LIN {X 0,Y 488.808,Z 370.599,A -85,B 0,C 180,E1 -6488.267,E2 -6488.267} C_VEL
LIN {X 0,Y 488.82,Z 370.594,A -85,B 0,C 180,E1 -6491.612,E2 -6491.612} C_VEL
LIN {X 0,Y 488.751,Z 370.602,A -85,B 0,C 180,E1 -6495.001,E2 -6495.001} C_VEL
LIN {X 0,Y 488.744,Z 370.605,A -85,B 0,C 180,E1 -6498.443,E2 -6498.443} C_VEL
LIN {X 0,Y 488.732,Z 370.603,A -85,B 0,C 180,E1 -6501.07,E2 -6501.07} C_VEL
LIN {X 0,Y 488.706,Z 370.612,A -85,B 0,C 180,E1 -6503.745,E2 -6503.745} C_VEL
LIN {X 0,Y 488.789,Z 370.596,A -85,B 0,C 180,E1 -6506.946,E2 -6506.946} C_VEL
LIN {X 0,Y 488.71,Z 370.607,A -85,B 0,C 180,E1 -6510.366,E2 -6510.366} C_VEL
LIN {X 0,Y 488.727,Z 370.609,A -85,B 0,C 180,E1 -6513.485,E2 -6513.485} C_VEL
LIN {X 0,Y 488.681,Z 370.609,A -85,B 0,C 180,E1 -6516.357,E2 -6516.357} C_VEL
LIN {X 0,Y 488.694,Z 370.613,A -85,B 0,C 180,E1 -6519.255,E2 -6519.255} C_VEL
LIN {X 0,Y 488.716,Z 370.609,A -85,B 0,C 180,E1 -6521.603,E2 -6521.603} C_VEL
LIN {X 0,Y 488.705,Z 370.608,A -85,B 0,C 180,E1 -6524.802,E2 -6524.802} C_VEL
LIN {X 0,Y 488.689,Z 370.612,A -85,B 0,C 180,E1 -6527.476,E2 -6527.476} C_VEL
LIN {X 0,Y 488.727,Z 370.605,A -85,B 0,C 180,E1 -6529.678,E2 -6529.678} C_VEL
LIN {X 0,Y 488.678,Z 370.615,A -85,B 0,C 180,E1 -6532.843,E2 -6532.843} C_VEL
LIN {X 0,Y 488.731,Z 370.604,A -85,B 0,C 180,E1 -6535.889,E2 -6535.889} C_VEL
LIN {X 0,Y 488.715,Z 370.612,A -85,B 0,C 180,E1 -6538.823,E2 -6538.823} C_VEL
LIN {X 0,Y 488.745,Z 370.603,A -85,B 0,C 180,E1 -6541.673,E2 -6541.673} C_VEL
LIN {X 0,Y 488.752,Z 370.607,A -85,B 0,C 180,E1 -6544.446,E2 -6544.446} C_VEL
LIN {X 0,Y 488.799,Z 370.776,A -85,B 0,C 180,E1 -6544.889,E2 -6544.889} C_VEL
LIN {X 0,Y 490.72,Z 381.32,A -85,B 0,C 180,E1 -6546.858,E2 -6546.858} C_VEL
LIN {X 0,Y 490.125,Z 397.445,A -85,B 0,C 180,E1 -6549.653,E2 -6549.653} C_VEL
LIN {X 0,Y 489.515,Z 415.125,A -85,B 0,C 180,E1 -6552.669,E2 -6552.669} C_VEL
LIN {X 0,Y 489.298,Z 421.438,A -85,B 0,C 180,E1 -6553.737,E2 -6553.737} C_VEL
LIN {X 0,Y 491.719,Z 437.9,A -85,B 0,C 180,E1 -6554.068,E2 -6554.068} C_VEL
LIN {X 0,Y 491.078,Z 529.428,A -85,B 0,C 180,E1 -6555.444,E2 -6555.444} C_VEL
LIN {X 0,Y 490.774,Z 542.701,A -85,B 0,C 180,E1 -6555.806,E2 -6555.806} C_VEL
LIN {X 0,Y 490.402,Z 555.445,A -85,B 0,C 180,E1 -6556.323,E2 -6556.323} C_VEL
LIN {X 0,Y 490.037,Z 567.098,A -85,B 0,C 180,E1 -6556.967,E2 -6556.967} C_VEL
LIN {X 0,Y 489.578,Z 578.466,A -85,B 0,C 180,E1 -6557.777,E2 -6557.777} C_VEL
LIN {X 0,Y 489.234,Z 588.982,A -85,B 0,C 180,E1 -6558.714,E2 -6558.714} C_VEL
LIN {X 0,Y 488.855,Z 597.575,A -85,B 0,C 180,E1 -6559.649,E2 -6559.649} C_VEL
LIN {X 0,Y 488.555,Z 605.502,A -85,B 0,C 180,E1 -6560.688,E2 -6560.688} C_VEL
LIN {X 0,Y 488.289,Z 613.245,A -85,B 0,C 180,E1 -6561.934,E2 -6561.934} C_VEL
LIN {X 0,Y 488.068,Z 620.369,A -85,B 0,C 180,E1 -6563.386,E2 -6563.386} C_VEL
LIN {X 0,Y 488.022,Z 625.112,A -85,B 0,C 180,E1 -6564.63,E2 -6564.63} C_VEL
LIN {X 0,Y 487.927,Z 628.733,A -85,B 0,C 180,E1 -6565.871,E2 -6565.871} C_VEL
LIN {X 0,Y 487.964,Z 630.602,A -85,B 0,C 180,E1 -6566.698,E2 -6566.698} C_VEL
LIN {X 0,Y 487.908,Z 632.001,A -85,B 0,C 180,E1 -6567.524,E2 -6567.524} C_VEL
LIN {X 0,Y 487.89,Z 632.998,A -85,B 0,C 180,E1 -6568.35,E2 -6568.35} C_VEL
LIN {X 0,Y 487.819,Z 633.817,A -85,B 0,C 180,E1 -6570.001,E2 -6570.001} C_VEL
LIN {X 0,Y 487.891,Z 632.984,A -85,B 0,C 180,E1 -6571.652,E2 -6571.652} C_VEL
LIN {X 0,Y 487.909,Z 631.98,A -85,B 0,C 180,E1 -6572.478,E2 -6572.478} C_VEL
LIN {X 0,Y 487.965,Z 630.574,A -85,B 0,C 180,E1 -6573.304,E2 -6573.304} C_VEL
LIN {X 0,Y 487.921,Z 627.615,A -85,B 0,C 180,E1 -6574.545,E2 -6574.545} C_VEL
LIN {X 0,Y 488.033,Z 623.616,A -85,B 0,C 180,E1 -6575.787,E2 -6575.787} C_VEL
LIN {X 0,Y 488.184,Z 617.461,A -85,B 0,C 180,E1 -6577.238,E2 -6577.238} C_VEL
LIN {X 0,Y 488.365,Z 610.737,A -85,B 0,C 180,E1 -6578.483,E2 -6578.483} C_VEL
LIN {X 0,Y 488.663,Z 602.397,A -85,B 0,C 180,E1 -6579.73,E2 -6579.73} C_VEL
LIN {X 0,Y 489.003,Z 593.832,A -85,B 0,C 180,E1 -6580.769,E2 -6580.769} C_VEL
LIN {X 0,Y 489.456,Z 583.255,A -85,B 0,C 180,E1 -6581.808,E2 -6581.808} C_VEL
LIN {X 0,Y 489.761,Z 572.902,A -85,B 0,C 180,E1 -6582.633,E2 -6582.633} C_VEL
LIN {X 0,Y 490.209,Z 561.27,A -85,B 0,C 180,E1 -6583.368,E2 -6583.368} C_VEL
LIN {X 0,Y 490.569,Z 549.352,A -85,B 0,C 180,E1 -6583.938,E2 -6583.938} C_VEL
LIN {X 0,Y 490.887,Z 535.598,A -85,B 0,C 180,E1 -6584.405,E2 -6584.405} C_VEL
LIN {X 0,Y 491.16,Z 523.133,A -85,B 0,C 180,E1 -6584.661,E2 -6584.661} C_VEL
LIN {X 0,Y 491.597,Z 435.781,A -85,B 0,C 180,E1 -6585.966,E2 -6585.966} C_VEL
LIN {X 0,Y 489.275,Z 421.167,A -85,B 0,C 180,E1 -6586.268,E2 -6586.268} C_VEL
LIN {X 0,Y 489.841,Z 403.479,A -85,B 0,C 180,E1 -6589.269,E2 -6589.269} C_VEL
LIN {X 0,Y 490.421,Z 388.337,A -85,B 0,C 180,E1 -6591.877,E2 -6591.877} C_VEL
LIN {X 0,Y 490.673,Z 381.092,A -85,B 0,C 180,E1 -6593.141,E2 -6593.141} C_VEL
LIN {X 0,Y 488.772,Z 370.605,A -85,B 0,C 180,E1 -6595.114,E2 -6595.114} C_VEL
LIN {X 0,Y 488.752,Z 370.608,A -85,B 0,C 180,E1 -6597.397,E2 -6597.397} C_VEL
LIN {X 0,Y 488.715,Z 370.608,A -85,B 0,C 180,E1 -6600.363,E2 -6600.363} C_VEL
LIN {X 0,Y 488.741,Z 370.607,A -85,B 0,C 180,E1 -6603.485,E2 -6603.485} C_VEL
LIN {X 0,Y 488.688,Z 370.61,A -85,B 0,C 180,E1 -6606.355,E2 -6606.355} C_VEL
LIN {X 0,Y 488.707,Z 370.614,A -85,B 0,C 180,E1 -6609.255,E2 -6609.255} C_VEL
LIN {X 0,Y 488.712,Z 370.609,A -85,B 0,C 180,E1 -6611.6,E2 -6611.6} C_VEL
LIN {X 0,Y 488.718,Z 370.611,A -85,B 0,C 180,E1 -6614.802,E2 -6614.802} C_VEL
LIN {X 0,Y 488.697,Z 370.609,A -85,B 0,C 180,E1 -6617.475,E2 -6617.475} C_VEL
LIN {X 0,Y 488.738,Z 370.6,A -85,B 0,C 180,E1 -6619.677,E2 -6619.677} C_VEL
LIN {X 0,Y 488.684,Z 370.613,A -85,B 0,C 180,E1 -6622.841,E2 -6622.841} C_VEL
LIN {X 0,Y 488.736,Z 370.6,A -85,B 0,C 180,E1 -6625.887,E2 -6625.887} C_VEL
LIN {X 0,Y 488.698,Z 370.61,A -85,B 0,C 180,E1 -6628.821,E2 -6628.821} C_VEL
LIN {X 0,Y 488.749,Z 370.6,A -85,B 0,C 180,E1 -6631.671,E2 -6631.671} C_VEL
LIN {X 0,Y 488.732,Z 370.606,A -85,B 0,C 180,E1 -6634.443,E2 -6634.443} C_VEL
LIN {X 0,Y 488.727,Z 370.601,A -85,B 0,C 180,E1 -6637.153,E2 -6637.153} C_VEL
LIN {X 0,Y 488.731,Z 370.604,A -85,B 0,C 180,E1 -6639.811,E2 -6639.811} C_VEL
LIN {X 0,Y 488.735,Z 370.607,A -85,B 0,C 180,E1 -6642.423,E2 -6642.423} C_VEL
LIN {X 0,Y 488.768,Z 370.595,A -85,B 0,C 180,E1 -6645,E2 -6645} C_VEL
LIN {X 0,Y 488.811,Z 370.597,A -85,B 0,C 180,E1 -6648.388,E2 -6648.388} C_VEL
LIN {X 0,Y 488.823,Z 370.593,A -85,B 0,C 180,E1 -6651.734,E2 -6651.734} C_VEL
LIN {X 0,Y 488.861,Z 370.592,A -85,B 0,C 180,E1 -6654.224,E2 -6654.224} C_VEL
LIN {X 0,Y 488.967,Z 370.571,A -85,B 0,C 180,E1 -6657.529,E2 -6657.529} C_VEL
LIN {X 0,Y 488.94,Z 370.576,A -85,B 0,C 180,E1 -6660.824,E2 -6660.824} C_VEL
LIN {X 0,Y 488.967,Z 370.576,A -85,B 0,C 180,E1 -6662.471,E2 -6662.471} C_VEL
LIN {X 0,Y 488.861,Z 370.593,A -85,B 0,C 180,E1 -6665.776,E2 -6665.776} C_VEL
LIN {X 0,Y 488.823,Z 370.595,A -85,B 0,C 180,E1 -6668.266,E2 -6668.266} C_VEL
LIN {X 0,Y 488.812,Z 370.599,A -85,B 0,C 180,E1 -6671.612,E2 -6671.612} C_VEL
LIN {X 0,Y 488.768,Z 370.599,A -85,B 0,C 180,E1 -6675,E2 -6675} C_VEL
LIN {X 0,Y 488.761,Z 370.601,A -85,B 0,C 180,E1 -6678.442,E2 -6678.442} C_VEL
LIN {X 0,Y 488.713,Z 370.608,A -85,B 0,C 180,E1 -6681.071,E2 -6681.071} C_VEL
LIN {X 0,Y 488.686,Z 370.613,A -85,B 0,C 180,E1 -6683.746,E2 -6683.746} C_VEL
LIN {X 0,Y 488.798,Z 370.599,A -85,B 0,C 180,E1 -6686.943,E2 -6686.943} C_VEL
LIN {X 0,Y 488.752,Z 370.657,A -85,B 0,C 180,E1 -6690.491,E2 -6690.491} C_VEL
LIN {X 0,Y 489.968,Z 378.441,A -85,B 0,C 180,E1 -6692.189,E2 -6692.189} C_VEL
LIN {X 0,Y 489.5,Z 392.493,A -85,B 0,C 180,E1 -6695.076,E2 -6695.076} C_VEL
LIN {X 0,Y 489.419,Z 395.959,A -85,B 0,C 180,E1 -6695.783,E2 -6695.783} C_VEL
LIN {X 0,Y 491.819,Z 408.886,A -85,B 0,C 180,E1 -6696.08,E2 -6696.08} C_VEL
LIN {X 0,Y 491.092,Z 503.283,A -85,B 0,C 180,E1 -6697.509,E2 -6697.509} C_VEL
LIN {X 0,Y 490.847,Z 516.801,A -85,B 0,C 180,E1 -6697.89,E2 -6697.89} C_VEL
LIN {X 0,Y 490.536,Z 529.465,A -85,B 0,C 180,E1 -6698.421,E2 -6698.421} C_VEL
LIN {X 0,Y 490.143,Z 541.603,A -85,B 0,C 180,E1 -6699.117,E2 -6699.117} C_VEL
LIN {X 0,Y 489.713,Z 553.194,A -85,B 0,C 180,E1 -6699.972,E2 -6699.972} C_VEL
LIN {X 0,Y 489.32,Z 563.013,A -85,B 0,C 180,E1 -6700.877,E2 -6700.877} C_VEL
LIN {X 0,Y 488.97,Z 571.319,A -85,B 0,C 180,E1 -6701.808,E2 -6701.808} C_VEL
LIN {X 0,Y 488.651,Z 579.931,A -85,B 0,C 180,E1 -6702.989,E2 -6702.989} C_VEL
LIN {X 0,Y 488.392,Z 586.848,A -85,B 0,C 180,E1 -6704.154,E2 -6704.154} C_VEL
LIN {X 0,Y 488.333,Z 588.767,A -85,B 0,C 180,E1 -6704.521,E2 -6704.521} C_VEL
LIN {X 0,Y 487.535,Z 591.685,A -85,B 0,C 180,E1 -6705.122,E2 -6705.122} C_VEL
LIN {X 0,Y 484.558,Z 595.97,A -85,B 0,C 180,E1 -6706.116,E2 -6706.116} C_VEL
LIN {X 0,Y 481.618,Z 599.569,A -85,B 0,C 180,E1 -6707.156,E2 -6707.156} C_VEL
LIN {X 0,Y 480.887,Z 601.351,A -85,B 0,C 180,E1 -6707.822,E2 -6707.822} C_VEL
LIN {X 0,Y 480.726,Z 604.611,A -85,B 0,C 180,E1 -6709.484,E2 -6709.484} C_VEL
LIN {X 0,Y 480.705,Z 606.164,A -85,B 0,C 180,E1 -6711.047,E2 -6711.047} C_VEL
LIN {X 0,Y 480.715,Z 606.453,A -85,B 0,C 180,E1 -6712.137,E2 -6712.137} C_VEL
LIN {X 0,Y 480.677,Z 605.821,A -85,B 0,C 180,E1 -6713.529,E2 -6713.529} C_VEL
LIN {X 0,Y 480.794,Z 604.043,A -85,B 0,C 180,E1 -6714.943,E2 -6714.943} C_VEL
LIN {X 0,Y 480.893,Z 600.95,A -85,B 0,C 180,E1 -6716.411,E2 -6716.411} C_VEL
LIN {X 0,Y 481.023,Z 596.321,A -85,B 0,C 180,E1 -6717.932,E2 -6717.932} C_VEL
LIN {X 0,Y 481.212,Z 590.902,A -85,B 0,C 180,E1 -6719.257,E2 -6719.257} C_VEL
LIN {X 0,Y 481.466,Z 584.62,A -85,B 0,C 180,E1 -6720.479,E2 -6720.479} C_VEL
LIN {X 0,Y 481.782,Z 576.867,A -85,B 0,C 180,E1 -6721.699,E2 -6721.699} C_VEL
LIN {X 0,Y 482.092,Z 568.452,A -85,B 0,C 180,E1 -6722.782,E2 -6722.782} C_VEL
LIN {X 0,Y 482.56,Z 558.14,A -85,B 0,C 180,E1 -6723.859,E2 -6723.859} C_VEL
LIN {X 0,Y 483.058,Z 547.031,A -85,B 0,C 180,E1 -6724.78,E2 -6724.78} C_VEL
LIN {X 0,Y 483.414,Z 535.814,A -85,B 0,C 180,E1 -6725.521,E2 -6725.521} C_VEL
LIN {X 0,Y 483.745,Z 525.027,A -85,B 0,C 180,E1 -6726.075,E2 -6726.075} C_VEL
LIN {X 0,Y 484.059,Z 512.697,A -85,B 0,C 180,E1 -6726.542,E2 -6726.542} C_VEL
LIN {X 0,Y 484.242,Z 500.008,A -85,B 0,C 180,E1 -6726.853,E2 -6726.853} C_VEL
LIN {X 0,Y 484.866,Z 409.068,A -85,B 0,C 180,E1 -6728.237,E2 -6728.237} C_VEL
LIN {X 0,Y 482.372,Z 395.878,A -85,B 0,C 180,E1 -6728.54,E2 -6728.54} C_VEL
LIN {X 0,Y 482.945,Z 380.242,A -85,B 0,C 180,E1 -6731.766,E2 -6731.766} C_VEL
LIN {X 0,Y 482.615,Z 376.203,A -85,B 0,C 180,E1 -6732.63,E2 -6732.63} C_VEL
LIN {X 0,Y 481.754,Z 371.477,A -85,B 0,C 180,E1 -6733.69,E2 -6733.69} C_VEL
LIN {X 0,Y 481.701,Z 371.485,A -85,B 0,C 180,E1 -6736.499,E2 -6736.499} C_VEL
LIN {X 0,Y 481.713,Z 371.479,A -85,B 0,C 180,E1 -6739.066,E2 -6739.066} C_VEL
LIN {X 0,Y 481.768,Z 371.469,A -85,B 0,C 180,E1 -6741.611,E2 -6741.611} C_VEL
LIN {X 0,Y 481.782,Z 371.469,A -85,B 0,C 180,E1 -6744.978,E2 -6744.978} C_VEL
LIN {X 0,Y 481.933,Z 371.449,A -85,B 0,C 180,E1 -6747.492,E2 -6747.492} C_VEL
LIN {X 0,Y 481.909,Z 371.454,A -85,B 0,C 180,E1 -6750.835,E2 -6750.835} C_VEL
LIN {X 0,Y 481.932,Z 371.454,A -85,B 0,C 180,E1 -6752.506,E2 -6752.506} C_VEL
LIN {X 0,Y 481.819,Z 371.466,A -85,B 0,C 180,E1 -6755.859,E2 -6755.859} C_VEL
LIN {X 0,Y 481.764,Z 371.475,A -85,B 0,C 180,E1 -6758.387,E2 -6758.387} C_VEL
LIN {X 0,Y 481.753,Z 371.475,A -85,B 0,C 180,E1 -6761.784,E2 -6761.784} C_VEL
LIN {X 0,Y 481.744,Z 371.472,A -85,B 0,C 180,E1 -6765.223,E2 -6765.223} C_VEL
LIN {X 0,Y 481.713,Z 371.477,A -85,B 0,C 180,E1 -6768.72,E2 -6768.72} C_VEL
LIN {X 0,Y 481.645,Z 371.486,A -85,B 0,C 180,E1 -6771.393,E2 -6771.393} C_VEL
LIN {X 0,Y 481.658,Z 371.488,A -85,B 0,C 180,E1 -6774.113,E2 -6774.113} C_VEL
LIN {X 0,Y 481.746,Z 371.473,A -85,B 0,C 180,E1 -6777.138,E2 -6777.138} C_VEL
LIN {X 0,Y 481.686,Z 371.488,A -85,B 0,C 180,E1 -6779.739,E2 -6779.739} C_VEL
LIN {X 0,Y 481.671,Z 371.481,A -85,B 0,C 180,E1 -6782.673,E2 -6782.673} C_VEL
LIN {X 0,Y 481.64,Z 371.493,A -85,B 0,C 180,E1 -6785.708,E2 -6785.708} C_VEL
LIN {X 0,Y 481.712,Z 371.481,A -85,B 0,C 180,E1 -6789.353,E2 -6789.353} C_VEL
LIN {X 0,Y 481.649,Z 371.485,A -85,B 0,C 180,E1 -6792.159,E2 -6792.159} C_VEL
LIN {X 0,Y 481.654,Z 371.491,A -85,B 0,C 180,E1 -6795.542,E2 -6795.542} C_VEL
LIN {X 0,Y 481.728,Z 371.587,A -85,B 0,C 180,E1 -6796.992,E2 -6796.992} C_VEL
LIN {X 0,Y 482.654,Z 377.903,A -85,B 0,C 180,E1 -6798.249,E2 -6798.249} C_VEL
LIN {X 0,Y 482.331,Z 393.362,A -85,B 0,C 180,E1 -6801.204,E2 -6801.204} C_VEL
LIN {X 0,Y 482.281,Z 395.35,A -85,B 0,C 180,E1 -6801.58,E2 -6801.58} C_VEL
LIN {X 0,Y 484.868,Z 410.274,A -85,B 0,C 180,E1 -6801.912,E2 -6801.912} C_VEL
LIN {X 0,Y 484.055,Z 502.974,A -85,B 0,C 180,E1 -6803.376,E2 -6803.376} C_VEL
LIN {X 0,Y 483.82,Z 514.928,A -85,B 0,C 180,E1 -6803.705,E2 -6803.705} C_VEL
LIN {X 0,Y 483.542,Z 527.078,A -85,B 0,C 180,E1 -6804.196,E2 -6804.196} C_VEL
LIN {X 0,Y 483.188,Z 538.287,A -85,B 0,C 180,E1 -6804.806,E2 -6804.806} C_VEL
LIN {X 0,Y 482.775,Z 549.847,A -85,B 0,C 180,E1 -6805.611,E2 -6805.611} C_VEL
LIN {X 0,Y 482.351,Z 560.102,A -85,B 0,C 180,E1 -6806.506,E2 -6806.506} C_VEL
LIN {X 0,Y 481.921,Z 570.355,A -85,B 0,C 180,E1 -6807.623,E2 -6807.623} C_VEL
LIN {X 0,Y 481.618,Z 579.109,A -85,B 0,C 180,E1 -6808.799,E2 -6808.799} C_VEL
LIN {X 0,Y 481.281,Z 586.3,A -85,B 0,C 180,E1 -6809.991,E2 -6809.991} C_VEL
LIN {X 0,Y 481.134,Z 592.238,A -85,B 0,C 180,E1 -6811.211,E2 -6811.211} C_VEL
LIN {X 0,Y 480.957,Z 597.537,A -85,B 0,C 180,E1 -6812.594,E2 -6812.594} C_VEL
LIN {X 0,Y 480.844,Z 601.545,A -85,B 0,C 180,E1 -6813.993,E2 -6813.993} C_VEL
LIN {X 0,Y 480.775,Z 603.639,A -85,B 0,C 180,E1 -6814.998,E2 -6814.998} C_VEL
LIN {X 0,Y 480.709,Z 604.92,A -85,B 0,C 180,E1 -6815.835,E2 -6815.835} C_VEL
LIN {X 0,Y 480.712,Z 606.065,A -85,B 0,C 180,E1 -6817.077,E2 -6817.077} C_VEL
LIN {X 0,Y 480.689,Z 606.282,A -85,B 0,C 180,E1 -6818.56,E2 -6818.56} C_VEL
LIN {X 0,Y 480.756,Z 605.793,A -85,B 0,C 180,E1 -6819.461,E2 -6819.461} C_VEL
LIN {X 0,Y 480.737,Z 604.831,A -85,B 0,C 180,E1 -6820.352,E2 -6820.352} C_VEL
LIN {X 0,Y 480.844,Z 602.28,A -85,B 0,C 180,E1 -6821.807,E2 -6821.807} C_VEL
LIN {X 0,Y 480.902,Z 599.178,A -85,B 0,C 180,E1 -6823.005,E2 -6823.005} C_VEL
LIN {X 0,Y 481.013,Z 594.732,A -85,B 0,C 180,E1 -6824.302,E2 -6824.302} C_VEL
LIN {X 0,Y 481.273,Z 588.866,A -85,B 0,C 180,E1 -6825.626,E2 -6825.626} C_VEL
LIN {X 0,Y 481.486,Z 581.582,A -85,B 0,C 180,E1 -6826.924,E2 -6826.924} C_VEL
LIN {X 0,Y 481.82,Z 573.626,A -85,B 0,C 180,E1 -6828.073,E2 -6828.073} C_VEL
LIN {X 0,Y 482.202,Z 564.181,A -85,B 0,C 180,E1 -6829.184,E2 -6829.184} C_VEL
LIN {X 0,Y 482.615,Z 554.003,A -85,B 0,C 180,E1 -6830.148,E2 -6830.148} C_VEL
LIN {X 0,Y 483.088,Z 542.602,A -85,B 0,C 180,E1 -6831.014,E2 -6831.014} C_VEL
LIN {X 0,Y 483.458,Z 531.132,A -85,B 0,C 180,E1 -6831.694,E2 -6831.694} C_VEL
LIN {X 0,Y 483.762,Z 517.949,A -85,B 0,C 180,E1 -6832.277,E2 -6832.277} C_VEL
LIN {X 0,Y 484.035,Z 505.763,A -85,B 0,C 180,E1 -6832.649,E2 -6832.649} C_VEL
LIN {X 0,Y 484.242,Z 484.353,A -85,B 0,C 180,E1 -6833.018,E2 -6833.018} C_VEL
LIN {X 0,Y 484.862,Z 409.135,A -85,B 0,C 180,E1 -6834.216,E2 -6834.216} C_VEL
LIN {X 0,Y 482.352,Z 395.683,A -85,B 0,C 180,E1 -6834.539,E2 -6834.539} C_VEL
LIN {X 0,Y 482.611,Z 379.888,A -85,B 0,C 180,E1 -6837.496,E2 -6837.496} C_VEL
LIN {X 0,Y 482.46,Z 375.431,A -85,B 0,C 180,E1 -6838.33,E2 -6838.33} C_VEL
LIN {X 0,Y 481.9,Z 371.461,A -85,B 0,C 180,E1 -6839.112,E2 -6839.112} C_VEL
LIN {X 0,Y 481.801,Z 371.469,A -85,B 0,C 180,E1 -6841.672,E2 -6841.672} C_VEL
LIN {X 0,Y 481.919,Z 371.46,A -85,B 0,C 180,E1 -6842.507,E2 -6842.507} C_VEL
LIN {X 0,Y 481.807,Z 371.47,A -85,B 0,C 180,E1 -6845.86,E2 -6845.86} C_VEL
LIN {X 0,Y 481.753,Z 371.478,A -85,B 0,C 180,E1 -6848.388,E2 -6848.388} C_VEL
LIN {X 0,Y 481.784,Z 371.472,A -85,B 0,C 180,E1 -6851.784,E2 -6851.784} C_VEL
LIN {X 0,Y 481.732,Z 371.476,A -85,B 0,C 180,E1 -6855.225,E2 -6855.225} C_VEL
LIN {X 0,Y 481.702,Z 371.48,A -85,B 0,C 180,E1 -6858.722,E2 -6858.722} C_VEL
LIN {X 0,Y 481.668,Z 371.485,A -85,B 0,C 180,E1 -6861.394,E2 -6861.394} C_VEL
LIN {X 0,Y 481.683,Z 371.485,A -85,B 0,C 180,E1 -6864.113,E2 -6864.113} C_VEL
LIN {X 0,Y 481.742,Z 371.475,A -85,B 0,C 180,E1 -6867.141,E2 -6867.141} C_VEL
LIN {X 0,Y 481.679,Z 371.487,A -85,B 0,C 180,E1 -6869.741,E2 -6869.741} C_VEL
LIN {X 0,Y 481.664,Z 371.484,A -85,B 0,C 180,E1 -6872.675,E2 -6872.675} C_VEL
LIN {X 0,Y 481.634,Z 371.493,A -85,B 0,C 180,E1 -6875.71,E2 -6875.71} C_VEL
LIN {X 0,Y 481.664,Z 371.485,A -85,B 0,C 180,E1 -6878.86,E2 -6878.86} C_VEL
LIN {X 0,Y 481.655,Z 371.486,A -85,B 0,C 180,E1 -6881.915,E2 -6881.915} C_VEL
LIN {X 0,Y 481.653,Z 371.484,A -85,B 0,C 180,E1 -6884.458,E2 -6884.458} C_VEL
LIN {X 0,Y 481.671,Z 371.486,A -85,B 0,C 180,E1 -6886.848,E2 -6886.848} C_VEL
LIN {X 0,Y 481.671,Z 371.483,A -85,B 0,C 180,E1 -6890.061,E2 -6890.061} C_VEL
LIN {X 0,Y 481.625,Z 371.492,A -85,B 0,C 180,E1 -6893.255,E2 -6893.255} C_VEL
LIN {X 0,Y 481.705,Z 371.481,A -85,B 0,C 180,E1 -6896.331,E2 -6896.331} C_VEL
LIN {X 0,Y 481.662,Z 371.486,A -85,B 0,C 180,E1 -6899.416,E2 -6899.416} C_VEL
LIN {X 0,Y 481.701,Z 371.482,A -85,B 0,C 180,E1 -6902.17,E2 -6902.17} C_VEL
LIN {X 0,Y 481.753,Z 371.589,A -85,B 0,C 180,E1 -6904.677,E2 -6904.677} C_VEL
LIN {X 0,Y 483.653,Z 381.843,A -85,B 0,C 180,E1 -6906.627,E2 -6906.627} C_VEL
LIN {X 0,Y 483.465,Z 390.788,A -85,B 0,C 180,E1 -6908.215,E2 -6908.215} C_VEL
LIN {X 0,Y 482.763,Z 409.881,A -85,B 0,C 180,E1 -6911.542,E2 -6911.542} C_VEL
LIN {X 0,Y 482.339,Z 421.377,A -85,B 0,C 180,E1 -6913.5,E2 -6913.5} C_VEL
LIN {X 0,Y 484.882,Z 438.54,A -85,B 0,C 180,E1 -6913.852,E2 -6913.852} C_VEL
LIN {X 0,Y 484.186,Z 530.163,A -85,B 0,C 180,E1 -6915.259,E2 -6915.259} C_VEL
LIN {X 0,Y 483.872,Z 543.124,A -85,B 0,C 180,E1 -6915.626,E2 -6915.626} C_VEL
LIN {X 0,Y 483.497,Z 555.141,A -85,B 0,C 180,E1 -6916.124,E2 -6916.124} C_VEL
LIN {X 0,Y 483.099,Z 566.506,A -85,B 0,C 180,E1 -6916.756,E2 -6916.756} C_VEL
LIN {X 0,Y 482.619,Z 578.258,A -85,B 0,C 180,E1 -6917.602,E2 -6917.602} C_VEL
LIN {X 0,Y 482.205,Z 588.738,A -85,B 0,C 180,E1 -6918.547,E2 -6918.547} C_VEL
LIN {X 0,Y 481.835,Z 597.343,A -85,B 0,C 180,E1 -6919.496,E2 -6919.496} C_VEL
LIN {X 0,Y 481.501,Z 605.278,A -85,B 0,C 180,E1 -6920.55,E2 -6920.55} C_VEL
LIN {X 0,Y 481.235,Z 613.031,A -85,B 0,C 180,E1 -6921.815,E2 -6921.815} C_VEL
LIN {X 0,Y 481.007,Z 620.161,A -85,B 0,C 180,E1 -6923.289,E2 -6923.289} C_VEL
LIN {X 0,Y 480.935,Z 624.907,A -85,B 0,C 180,E1 -6924.551,E2 -6924.551} C_VEL
LIN {X 0,Y 480.828,Z 628.53,A -85,B 0,C 180,E1 -6925.81,E2 -6925.81} C_VEL
LIN {X 0,Y 480.888,Z 630.402,A -85,B 0,C 180,E1 -6926.65,E2 -6926.65} C_VEL
LIN {X 0,Y 480.823,Z 631.801,A -85,B 0,C 180,E1 -6927.488,E2 -6927.488} C_VEL
LIN {X 0,Y 480.792,Z 632.798,A -85,B 0,C 180,E1 -6928.326,E2 -6928.326} C_VEL
LIN {X 0,Y 480.76,Z 633.404,A -85,B 0,C 180,E1 -6929.163,E2 -6929.163} C_VEL
LIN {X 0,Y 480.743,Z 633.617,A -85,B 0,C 180,E1 -6930.001,E2 -6930.001} C_VEL
LIN {X 0,Y 480.76,Z 633.396,A -85,B 0,C 180,E1 -6930.839,E2 -6930.839} C_VEL
LIN {X 0,Y 480.792,Z 632.781,A -85,B 0,C 180,E1 -6931.676,E2 -6931.676} C_VEL
LIN {X 0,Y 480.823,Z 631.776,A -85,B 0,C 180,E1 -6932.514,E2 -6932.514} C_VEL
LIN {X 0,Y 480.888,Z 630.368,A -85,B 0,C 180,E1 -6933.352,E2 -6933.352} C_VEL
LIN {X 0,Y 480.84,Z 627.406,A -85,B 0,C 180,E1 -6934.612,E2 -6934.612} C_VEL
LIN {X 0,Y 480.936,Z 623.403,A -85,B 0,C 180,E1 -6935.872,E2 -6935.872} C_VEL
LIN {X 0,Y 481.112,Z 617.242,A -85,B 0,C 180,E1 -6937.345,E2 -6937.345} C_VEL
LIN {X 0,Y 481.325,Z 610.514,A -85,B 0,C 180,E1 -6938.608,E2 -6938.608} C_VEL
LIN {X 0,Y 481.613,Z 602.166,A -85,B 0,C 180,E1 -6939.874,E2 -6939.874} C_VEL
LIN {X 0,Y 482.003,Z 593.593,A -85,B 0,C 180,E1 -6940.928,E2 -6940.928} C_VEL
LIN {X 0,Y 482.484,Z 583.029,A -85,B 0,C 180,E1 -6941.979,E2 -6941.979} C_VEL
LIN {X 0,Y 482.787,Z 573.518,A -85,B 0,C 180,E1 -6942.753,E2 -6942.753} C_VEL
LIN {X 0,Y 483.216,Z 562.787,A -85,B 0,C 180,E1 -6943.458,E2 -6943.458} C_VEL
LIN {X 0,Y 483.64,Z 550.357,A -85,B 0,C 180,E1 -6944.088,E2 -6944.088} C_VEL
LIN {X 0,Y 483.968,Z 537.116,A -85,B 0,C 180,E1 -6944.562,E2 -6944.562} C_VEL
LIN {X 0,Y 484.284,Z 524.332,A -85,B 0,C 180,E1 -6944.847,E2 -6944.847} C_VEL
LIN {X 0,Y 484.807,Z 436.74,A -85,B 0,C 180,E1 -6946.179,E2 -6946.179} C_VEL
LIN {X 0,Y 482.27,Z 420.816,A -85,B 0,C 180,E1 -6946.538,E2 -6946.538} C_VEL
LIN {X 0,Y 482.916,Z 403.311,A -85,B 0,C 180,E1 -6949.557,E2 -6949.557} C_VEL
LIN {X 0,Y 483.599,Z 386.93,A -85,B 0,C 180,E1 -6952.427,E2 -6952.427} C_VEL
LIN {X 0,Y 483.635,Z 381.616,A -85,B 0,C 180,E1 -6953.377,E2 -6953.377} C_VEL
LIN {X 0,Y 481.724,Z 371.482,A -85,B 0,C 180,E1 -6955.353,E2 -6955.353} C_VEL
LIN {X 0,Y 481.706,Z 371.485,A -85,B 0,C 180,E1 -6957.833,E2 -6957.833} C_VEL
LIN {X 0,Y 481.651,Z 371.489,A -85,B 0,C 180,E1 -6960.712,E2 -6960.712} C_VEL
LIN {X 0,Y 481.702,Z 371.481,A -85,B 0,C 180,E1 -6963.734,E2 -6963.734} C_VEL
LIN {X 0,Y 481.631,Z 371.492,A -85,B 0,C 180,E1 -6966.747,E2 -6966.747} C_VEL
LIN {X 0,Y 481.682,Z 371.483,A -85,B 0,C 180,E1 -6969.941,E2 -6969.941} C_VEL
LIN {X 0,Y 481.645,Z 371.492,A -85,B 0,C 180,E1 -6973.3,E2 -6973.3} C_VEL
LIN {X 0,Y 481.664,Z 371.485,A -85,B 0,C 180,E1 -6975.641,E2 -6975.641} C_VEL
LIN {X 0,Y 481.662,Z 371.489,A -85,B 0,C 180,E1 -6978.959,E2 -6978.959} C_VEL
LIN {X 0,Y 481.659,Z 371.484,A -85,B 0,C 180,E1 -6981.993,E2 -6981.993} C_VEL
LIN {X 0,Y 481.694,Z 371.479,A -85,B 0,C 180,E1 -6985.318,E2 -6985.318} C_VEL
LIN {X 0,Y 481.651,Z 371.488,A -85,B 0,C 180,E1 -6988.312,E2 -6988.312} C_VEL
LIN {X 0,Y 481.704,Z 371.48,A -85,B 0,C 180,E1 -6991.219,E2 -6991.219} C_VEL
LIN {X 0,Y 481.695,Z 371.477,A -85,B 0,C 180,E1 -6994.042,E2 -6994.042} C_VEL
LIN {X 0,Y 481.68,Z 371.482,A -85,B 0,C 180,E1 -6996.812,E2 -6996.812} C_VEL
LIN {X 0,Y 481.701,Z 371.478,A -85,B 0,C 180,E1 -6999.503,E2 -6999.503} C_VEL
LIN {X 0,Y 481.71,Z 371.478,A -85,B 0,C 180,E1 -7002.159,E2 -7002.159} C_VEL
LIN {X 0,Y 481.748,Z 371.471,A -85,B 0,C 180,E1 -7004.776,E2 -7004.776} C_VEL
LIN {X 0,Y 481.757,Z 371.478,A -85,B 0,C 180,E1 -7008.215,E2 -7008.215} C_VEL
LIN {X 0,Y 481.768,Z 371.471,A -85,B 0,C 180,E1 -7011.612,E2 -7011.612} C_VEL
LIN {X 0,Y 481.822,Z 371.467,A -85,B 0,C 180,E1 -7014.14,E2 -7014.14} C_VEL
LIN {X 0,Y 481.934,Z 371.447,A -85,B 0,C 180,E1 -7017.493,E2 -7017.493} C_VEL
LIN {X 0,Y 481.892,Z 371.453,A -85,B 0,C 180,E1 -7020.836,E2 -7020.836} C_VEL
LIN {X 0,Y 481.934,Z 371.451,A -85,B 0,C 180,E1 -7022.508,E2 -7022.508} C_VEL
LIN {X 0,Y 481.822,Z 371.471,A -85,B 0,C 180,E1 -7025.86,E2 -7025.86} C_VEL
LIN {X 0,Y 481.769,Z 371.473,A -85,B 0,C 180,E1 -7028.388,E2 -7028.388} C_VEL
LIN {X 0,Y 481.757,Z 371.478,A -85,B 0,C 180,E1 -7031.785,E2 -7031.785} C_VEL
LIN {X 0,Y 481.749,Z 371.475,A -85,B 0,C 180,E1 -7035.224,E2 -7035.224} C_VEL
LIN {X 0,Y 481.718,Z 371.478,A -85,B 0,C 180,E1 -7038.722,E2 -7038.722} C_VEL
LIN {X 0,Y 481.652,Z 371.49,A -85,B 0,C 180,E1 -7041.395,E2 -7041.395} C_VEL
LIN {X 0,Y 481.667,Z 371.487,A -85,B 0,C 180,E1 -7044.114,E2 -7044.114} C_VEL
LIN {X 0,Y 481.753,Z 371.478,A -85,B 0,C 180,E1 -7047.139,E2 -7047.139} C_VEL
LIN {X 0,Y 481.717,Z 371.632,A -85,B 0,C 180,E1 -7050.322,E2 -7050.322} C_VEL
LIN {X 0,Y 483.031,Z 379.195,A -85,B 0,C 180,E1 -7052.006,E2 -7052.006} C_VEL
LIN {X 0,Y 482.536,Z 393.432,A -85,B 0,C 180,E1 -7054.97,E2 -7054.97} C_VEL
LIN {X 0,Y 482.46,Z 396.504,A -85,B 0,C 180,E1 -7055.56,E2 -7055.56} C_VEL
LIN {X 0,Y 485.013,Z 410.532,A -85,B 0,C 180,E1 -7055.871,E2 -7055.871} C_VEL
LIN {X 0,Y 484.228,Z 503.506,A -85,B 0,C 180,E1 -7057.301,E2 -7057.301} C_VEL
LIN {X 0,Y 483.952,Z 517.202,A -85,B 0,C 180,E1 -7057.694,E2 -7057.694} C_VEL
LIN {X 0,Y 483.657,Z 529.479,A -85,B 0,C 180,E1 -7058.216,E2 -7058.216} C_VEL
LIN {X 0,Y 483.244,Z 541.606,A -85,B 0,C 180,E1 -7058.918,E2 -7058.918} C_VEL
LIN {X 0,Y 482.771,Z 552.69,A -85,B 0,C 180,E1 -7059.74,E2 -7059.74} C_VEL
LIN {X 0,Y 482.324,Z 563.419,A -85,B 0,C 180,E1 -7060.737,E2 -7060.737} C_VEL
LIN {X 0,Y 481.94,Z 572.227,A -85,B 0,C 180,E1 -7061.752,E2 -7061.752} C_VEL
LIN {X 0,Y 481.624,Z 580.285,A -85,B 0,C 180,E1 -7062.882,E2 -7062.882} C_VEL
LIN {X 0,Y 481.34,Z 587.5,A -85,B 0,C 180,E1 -7064.124,E2 -7064.124} C_VEL
LIN {X 0,Y 481.119,Z 593.782,A -85,B 0,C 180,E1 -7065.478,E2 -7065.478} C_VEL
LIN {X 0,Y 480.954,Z 598.942,A -85,B 0,C 180,E1 -7066.94,E2 -7066.94} C_VEL
LIN {X 0,Y 480.887,Z 601.351,A -85,B 0,C 180,E1 -7067.822,E2 -7067.822} C_VEL
LIN {X 0,Y 480.15,Z 602.918,A -85,B 0,C 180,E1 -7068.496,E2 -7068.496} C_VEL
LIN {X 0,Y 477.204,Z 604.948,A -85,B 0,C 180,E1 -7069.603,E2 -7069.603} C_VEL
LIN {X 0,Y 474.747,Z 606.05,A -85,B 0,C 180,E1 -7070.505,E2 -7070.505} C_VEL
LIN {X 0,Y 473.69,Z 606.498,A -85,B 0,C 180,E1 -7071.208,E2 -7071.208} C_VEL
LIN {X 0,Y 473.601,Z 606.564,A -85,B 0,C 180,E1 -7071.447,E2 -7071.447} C_VEL
LIN {X 0,Y 473.624,Z 606.578,A -85,B 0,C 180,E1 -7072.526,E2 -7072.526} C_VEL
LIN {X 0,Y 473.611,Z 605.984,A -85,B 0,C 180,E1 -7073.588,E2 -7073.588} C_VEL
LIN {X 0,Y 473.675,Z 604.712,A -85,B 0,C 180,E1 -7074.691,E2 -7074.691} C_VEL
LIN {X 0,Y 473.789,Z 601.908,A -85,B 0,C 180,E1 -7076.169,E2 -7076.169} C_VEL
LIN {X 0,Y 473.918,Z 597.468,A -85,B 0,C 180,E1 -7077.732,E2 -7077.732} C_VEL
LIN {X 0,Y 474.138,Z 591.45,A -85,B 0,C 180,E1 -7079.285,E2 -7079.285} C_VEL
LIN {X 0,Y 474.459,Z 584.034,A -85,B 0,C 180,E1 -7080.736,E2 -7080.736} C_VEL
LIN {X 0,Y 474.796,Z 576.208,A -85,B 0,C 180,E1 -7081.961,E2 -7081.961} C_VEL
LIN {X 0,Y 475.163,Z 567.569,A -85,B 0,C 180,E1 -7083.065,E2 -7083.065} C_VEL
LIN {X 0,Y 475.603,Z 558.274,A -85,B 0,C 180,E1 -7084.034,E2 -7084.034} C_VEL
LIN {X 0,Y 476.156,Z 546.634,A -85,B 0,C 180,E1 -7085.006,E2 -7085.006} C_VEL
LIN {X 0,Y 476.544,Z 535.478,A -85,B 0,C 180,E1 -7085.745,E2 -7085.745} C_VEL
LIN {X 0,Y 476.885,Z 524.107,A -85,B 0,C 180,E1 -7086.326,E2 -7086.326} C_VEL
LIN {X 0,Y 477.201,Z 511.224,A -85,B 0,C 180,E1 -7086.798,E2 -7086.798} C_VEL
LIN {X 0,Y 477.428,Z 497.61,A -85,B 0,C 180,E1 -7087.11,E2 -7087.11} C_VEL
LIN {X 0,Y 478.025,Z 409.797,A -85,B 0,C 180,E1 -7088.462,E2 -7088.462} C_VEL
LIN {X 0,Y 475.414,Z 396.024,A -85,B 0,C 180,E1 -7088.791,E2 -7088.791} C_VEL
LIN {X 0,Y 475.999,Z 380.987,A -85,B 0,C 180,E1 -7091.936,E2 -7091.936} C_VEL
LIN {X 0,Y 474.787,Z 372.733,A -85,B 0,C 180,E1 -7093.759,E2 -7093.759} C_VEL
LIN {X 0,Y 474.724,Z 372.353,A -85,B 0,C 180,E1 -7093.852,E2 -7093.852} C_VEL
LIN {X 0,Y 474.707,Z 372.351,A -85,B 0,C 180,E1 -7097.723,E2 -7097.723} C_VEL
LIN {X 0,Y 474.711,Z 372.355,A -85,B 0,C 180,E1 -7100.626,E2 -7100.626} C_VEL
LIN {X 0,Y 474.709,Z 372.349,A -85,B 0,C 180,E1 -7103.197,E2 -7103.197} C_VEL
LIN {X 0,Y 474.752,Z 372.346,A -85,B 0,C 180,E1 -7104.903,E2 -7104.903} C_VEL
LIN {X 0,Y 474.899,Z 372.325,A -85,B 0,C 180,E1 -7107.454,E2 -7107.454} C_VEL
LIN {X 0,Y 474.916,Z 372.326,A -85,B 0,C 180,E1 -7109.999,E2 -7109.999} C_VEL
LIN {X 0,Y 474.898,Z 372.33,A -85,B 0,C 180,E1 -7112.543,E2 -7112.543} C_VEL
LIN {X 0,Y 474.782,Z 372.344,A -85,B 0,C 180,E1 -7115.946,E2 -7115.946} C_VEL
LIN {X 0,Y 474.729,Z 372.35,A -85,B 0,C 180,E1 -7118.512,E2 -7118.512} C_VEL
LIN {X 0,Y 474.707,Z 372.355,A -85,B 0,C 180,E1 -7121.961,E2 -7121.961} C_VEL
LIN {X 0,Y 474.703,Z 372.354,A -85,B 0,C 180,E1 -7125.776,E2 -7125.776} C_VEL
LIN {X 0,Y 474.665,Z 372.354,A -85,B 0,C 180,E1 -7129.009,E2 -7129.009} C_VEL
LIN {X 0,Y 474.589,Z 372.369,A -85,B 0,C 180,E1 -7131.728,E2 -7131.728} C_VEL
LIN {X 0,Y 474.638,Z 372.358,A -85,B 0,C 180,E1 -7134.493,E2 -7134.493} C_VEL
LIN {X 0,Y 474.697,Z 372.352,A -85,B 0,C 180,E1 -7137.337,E2 -7137.337} C_VEL
LIN {X 0,Y 474.608,Z 372.361,A -85,B 0,C 180,E1 -7140.81,E2 -7140.81} C_VEL
LIN {X 0,Y 474.635,Z 372.362,A -85,B 0,C 180,E1 -7143.983,E2 -7143.983} C_VEL
LIN {X 0,Y 474.572,Z 372.366,A -85,B 0,C 180,E1 -7146.899,E2 -7146.899} C_VEL
LIN {X 0,Y 474.648,Z 372.363,A -85,B 0,C 180,E1 -7149.65,E2 -7149.65} C_VEL
LIN {X 0,Y 474.63,Z 372.36,A -85,B 0,C 180,E1 -7152.931,E2 -7152.931} C_VEL
LIN {X 0,Y 474.611,Z 372.367,A -85,B 0,C 180,E1 -7155.895,E2 -7155.895} C_VEL
LIN {X 0,Y 474.672,Z 372.466,A -85,B 0,C 180,E1 -7156.866,E2 -7156.866} C_VEL
LIN {X 0,Y 475.602,Z 378.059,A -85,B 0,C 180,E1 -7157.986,E2 -7157.986} C_VEL
LIN {X 0,Y 475.437,Z 391.222,A -85,B 0,C 180,E1 -7160.533,E2 -7160.533} C_VEL
LIN {X 0,Y 475.307,Z 395.407,A -85,B 0,C 180,E1 -7161.334,E2 -7161.334} C_VEL
LIN {X 0,Y 478.028,Z 410.229,A -85,B 0,C 180,E1 -7161.68,E2 -7161.68} C_VEL
LIN {X 0,Y 477.162,Z 503.352,A -85,B 0,C 180,E1 -7163.182,E2 -7163.182} C_VEL
LIN {X 0,Y 476.901,Z 516.329,A -85,B 0,C 180,E1 -7163.553,E2 -7163.553} C_VEL
LIN {X 0,Y 476.548,Z 529.111,A -85,B 0,C 180,E1 -7164.103,E2 -7164.103} C_VEL
LIN {X 0,Y 476.159,Z 540.361,A -85,B 0,C 180,E1 -7164.748,E2 -7164.748} C_VEL
LIN {X 0,Y 475.723,Z 551.873,A -85,B 0,C 180,E1 -7165.592,E2 -7165.592} C_VEL
LIN {X 0,Y 475.274,Z 562.478,A -85,B 0,C 180,E1 -7166.576,E2 -7166.576} C_VEL
LIN {X 0,Y 474.859,Z 571.382,A -85,B 0,C 180,E1 -7167.587,E2 -7167.587} C_VEL
LIN {X 0,Y 474.571,Z 579.972,A -85,B 0,C 180,E1 -7168.78,E2 -7168.78} C_VEL
LIN {X 0,Y 474.214,Z 587.011,A -85,B 0,C 180,E1 -7169.988,E2 -7169.988} C_VEL
LIN {X 0,Y 474.037,Z 593.309,A -85,B 0,C 180,E1 -7171.334,E2 -7171.334} C_VEL
LIN {X 0,Y 473.856,Z 598.8,A -85,B 0,C 180,E1 -7172.856,E2 -7172.856} C_VEL
LIN {X 0,Y 473.755,Z 601.992,A -85,B 0,C 180,E1 -7174.047,E2 -7174.047} C_VEL
LIN {X 0,Y 473.635,Z 604.634,A -85,B 0,C 180,E1 -7175.451,E2 -7175.451} C_VEL
LIN {X 0,Y 473.601,Z 606.172,A -85,B 0,C 180,E1 -7176.929,E2 -7176.929} C_VEL
LIN {X 0,Y 473.601,Z 606.53,A -85,B 0,C 180,E1 -7178.223,E2 -7178.223} C_VEL
LIN {X 0,Y 473.644,Z 606.18,A -85,B 0,C 180,E1 -7179.192,E2 -7179.192} C_VEL
LIN {X 0,Y 473.659,Z 605.455,A -85,B 0,C 180,E1 -7180.046,E2 -7180.046} C_VEL
LIN {X 0,Y 473.745,Z 602.806,A -85,B 0,C 180,E1 -7181.697,E2 -7181.697} C_VEL
LIN {X 0,Y 473.839,Z 599.045,A -85,B 0,C 180,E1 -7183.188,E2 -7183.188} C_VEL
LIN {X 0,Y 473.968,Z 594.374,A -85,B 0,C 180,E1 -7184.535,E2 -7184.535} C_VEL
LIN {X 0,Y 474.269,Z 587.358,A -85,B 0,C 180,E1 -7186.066,E2 -7186.066} C_VEL
LIN {X 0,Y 474.535,Z 579.989,A -85,B 0,C 180,E1 -7187.338,E2 -7187.338} C_VEL
LIN {X 0,Y 474.89,Z 571.82,A -85,B 0,C 180,E1 -7188.475,E2 -7188.475} C_VEL
LIN {X 0,Y 475.305,Z 562.225,A -85,B 0,C 180,E1 -7189.564,E2 -7189.564} C_VEL
LIN {X 0,Y 475.768,Z 551.602,A -85,B 0,C 180,E1 -7190.541,E2 -7190.541} C_VEL
LIN {X 0,Y 476.232,Z 539.911,A -85,B 0,C 180,E1 -7191.388,E2 -7191.388} C_VEL
LIN {X 0,Y 476.637,Z 528.083,A -85,B 0,C 180,E1 -7192.054,E2 -7192.054} C_VEL
LIN {X 0,Y 476.937,Z 515.858,A -85,B 0,C 180,E1 -7192.565,E2 -7192.565} C_VEL
LIN {X 0,Y 477.209,Z 502.239,A -85,B 0,C 180,E1 -7192.941,E2 -7192.941} C_VEL
LIN {X 0,Y 478.092,Z 409.89,A -85,B 0,C 180,E1 -7194.451,E2 -7194.451} C_VEL
LIN {X 0,Y 475.397,Z 395.81,A -85,B 0,C 180,E1 -7194.805,E2 -7194.805} C_VEL
LIN {X 0,Y 475.697,Z 379.527,A -85,B 0,C 180,E1 -7197.883,E2 -7197.883} C_VEL
LIN {X 0,Y 474.868,Z 372.336,A -85,B 0,C 180,E1 -7199.284,E2 -7199.284} C_VEL
LIN {X 0,Y 474.885,Z 372.336,A -85,B 0,C 180,E1 -7202.545,E2 -7202.545} C_VEL
LIN {X 0,Y 474.769,Z 372.347,A -85,B 0,C 180,E1 -7205.948,E2 -7205.948} C_VEL
LIN {X 0,Y 474.718,Z 372.354,A -85,B 0,C 180,E1 -7208.514,E2 -7208.514} C_VEL
LIN {X 0,Y 474.729,Z 372.353,A -85,B 0,C 180,E1 -7211.962,E2 -7211.962} C_VEL
LIN {X 0,Y 474.691,Z 372.357,A -85,B 0,C 180,E1 -7215.777,E2 -7215.777} C_VEL
LIN {X 0,Y 474.655,Z 372.357,A -85,B 0,C 180,E1 -7219.011,E2 -7219.011} C_VEL
LIN {X 0,Y 474.635,Z 372.364,A -85,B 0,C 180,E1 -7221.727,E2 -7221.727} C_VEL
LIN {X 0,Y 474.66,Z 372.357,A -85,B 0,C 180,E1 -7224.493,E2 -7224.493} C_VEL
LIN {X 0,Y 474.689,Z 372.355,A -85,B 0,C 180,E1 -7227.339,E2 -7227.339} C_VEL
LIN {X 0,Y 474.601,Z 372.364,A -85,B 0,C 180,E1 -7230.812,E2 -7230.812} C_VEL
LIN {X 0,Y 474.629,Z 372.363,A -85,B 0,C 180,E1 -7233.985,E2 -7233.985} C_VEL
LIN {X 0,Y 474.567,Z 372.369,A -85,B 0,C 180,E1 -7236.901,E2 -7236.901} C_VEL
LIN {X 0,Y 474.62,Z 372.366,A -85,B 0,C 180,E1 -7239.649,E2 -7239.649} C_VEL
LIN {X 0,Y 474.628,Z 372.363,A -85,B 0,C 180,E1 -7242.933,E2 -7242.933} C_VEL
LIN {X 0,Y 474.609,Z 372.362,A -85,B 0,C 180,E1 -7245.897,E2 -7245.897} C_VEL
LIN {X 0,Y 474.626,Z 372.366,A -85,B 0,C 180,E1 -7249.041,E2 -7249.041} C_VEL
LIN {X 0,Y 474.605,Z 372.364,A -85,B 0,C 180,E1 -7251.705,E2 -7251.705} C_VEL
LIN {X 0,Y 474.626,Z 372.365,A -85,B 0,C 180,E1 -7254.727,E2 -7254.727} C_VEL
LIN {X 0,Y 474.634,Z 372.359,A -85,B 0,C 180,E1 -7257.789,E2 -7257.789} C_VEL
LIN {X 0,Y 474.63,Z 372.366,A -85,B 0,C 180,E1 -7260.884,E2 -7260.884} C_VEL
LIN {X 0,Y 474.665,Z 372.359,A -85,B 0,C 180,E1 -7263.63,E2 -7263.63} C_VEL
LIN {X 0,Y 474.705,Z 372.45,A -85,B 0,C 180,E1 -7264.47,E2 -7264.47} C_VEL
LIN {X 0,Y 476.811,Z 384.449,A -85,B 0,C 180,E1 -7266.78,E2 -7266.78} C_VEL
LIN {X 0,Y 476.168,Z 399.599,A -85,B 0,C 180,E1 -7269.481,E2 -7269.481} C_VEL
LIN {X 0,Y 475.523,Z 415.998,A -85,B 0,C 180,E1 -7272.365,E2 -7272.365} C_VEL
LIN {X 0,Y 475.362,Z 421.044,A -85,B 0,C 180,E1 -7273.246,E2 -7273.246} C_VEL
LIN {X 0,Y 478.064,Z 439.127,A -85,B 0,C 180,E1 -7273.631,E2 -7273.631} C_VEL
LIN {X 0,Y 477.33,Z 529.722,A -85,B 0,C 180,E1 -7275.043,E2 -7275.043} C_VEL
LIN {X 0,Y 476.976,Z 543.525,A -85,B 0,C 180,E1 -7275.44,E2 -7275.44} C_VEL
LIN {X 0,Y 476.531,Z 555.93,A -85,B 0,C 180,E1 -7275.972,E2 -7275.972} C_VEL
LIN {X 0,Y 476.098,Z 568.295,A -85,B 0,C 180,E1 -7276.698,E2 -7276.698} C_VEL
LIN {X 0,Y 475.598,Z 579.153,A -85,B 0,C 180,E1 -7277.512,E2 -7277.512} C_VEL
LIN {X 0,Y 475.182,Z 589.559,A -85,B 0,C 180,E1 -7278.484,E2 -7278.484} C_VEL
LIN {X 0,Y 474.749,Z 598.813,A -85,B 0,C 180,E1 -7279.553,E2 -7279.553} C_VEL
LIN {X 0,Y 474.367,Z 607.812,A -85,B 0,C 180,E1 -7280.837,E2 -7280.837} C_VEL
LIN {X 0,Y 474.074,Z 615.058,A -85,B 0,C 180,E1 -7282.119,E2 -7282.119} C_VEL
LIN {X 0,Y 473.876,Z 621.416,A -85,B 0,C 180,E1 -7283.552,E2 -7283.552} C_VEL
LIN {X 0,Y 473.829,Z 626.02,A -85,B 0,C 180,E1 -7284.895,E2 -7284.895} C_VEL
LIN {X 0,Y 473.734,Z 628.325,A -85,B 0,C 180,E1 -7285.747,E2 -7285.747} C_VEL
LIN {X 0,Y 473.795,Z 630.198,A -85,B 0,C 180,E1 -7286.6,E2 -7286.6} C_VEL
LIN {X 0,Y 473.741,Z 631.6,A -85,B 0,C 180,E1 -7287.45,E2 -7287.45} C_VEL
LIN {X 0,Y 473.688,Z 633.204,A -85,B 0,C 180,E1 -7289.151,E2 -7289.151} C_VEL
LIN {X 0,Y 473.669,Z 633.417,A -85,B 0,C 180,E1 -7290.001,E2 -7290.001} C_VEL
LIN {X 0,Y 473.688,Z 633.196,A -85,B 0,C 180,E1 -7290.851,E2 -7290.851} C_VEL
LIN {X 0,Y 473.741,Z 631.574,A -85,B 0,C 180,E1 -7292.552,E2 -7292.552} C_VEL
LIN {X 0,Y 473.795,Z 630.164,A -85,B 0,C 180,E1 -7293.403,E2 -7293.403} C_VEL
LIN {X 0,Y 473.763,Z 627.2,A -85,B 0,C 180,E1 -7294.681,E2 -7294.681} C_VEL
LIN {X 0,Y 473.843,Z 623.191,A -85,B 0,C 180,E1 -7295.96,E2 -7295.96} C_VEL
LIN {X 0,Y 474.024,Z 617.024,A -85,B 0,C 180,E1 -7297.455,E2 -7297.455} C_VEL
LIN {X 0,Y 474.287,Z 610.291,A -85,B 0,C 180,E1 -7298.737,E2 -7298.737} C_VEL
LIN {X 0,Y 474.584,Z 601.94,A -85,B 0,C 180,E1 -7300.022,E2 -7300.022} C_VEL
LIN {X 0,Y 474.999,Z 593.363,A -85,B 0,C 180,E1 -7301.091,E2 -7301.091} C_VEL
LIN {X 0,Y 475.498,Z 583.036,A -85,B 0,C 180,E1 -7302.136,E2 -7302.136} C_VEL
LIN {X 0,Y 475.858,Z 572.576,A -85,B 0,C 180,E1 -7302.995,E2 -7302.995} C_VEL
LIN {X 0,Y 476.364,Z 560.759,A -85,B 0,C 180,E1 -7303.764,E2 -7303.764} C_VEL
LIN {X 0,Y 476.792,Z 548.817,A -85,B 0,C 180,E1 -7304.349,E2 -7304.349} C_VEL
LIN {X 0,Y 477.18,Z 535.038,A -85,B 0,C 180,E1 -7304.828,E2 -7304.828} C_VEL
LIN {X 0,Y 477.448,Z 522.482,A -85,B 0,C 180,E1 -7305.092,E2 -7305.092} C_VEL
LIN {X 0,Y 477.979,Z 437.499,A -85,B 0,C 180,E1 -7306.405,E2 -7306.405} C_VEL
LIN {X 0,Y 475.271,Z 420.684,A -85,B 0,C 180,E1 -7306.778,E2 -7306.778} C_VEL
LIN {X 0,Y 475.917,Z 404.533,A -85,B 0,C 180,E1 -7309.609,E2 -7309.609} C_VEL
LIN {X 0,Y 476.674,Z 388.042,A -85,B 0,C 180,E1 -7312.542,E2 -7312.542} C_VEL
LIN {X 0,Y 476.728,Z 383.019,A -85,B 0,C 180,E1 -7313.457,E2 -7313.457} C_VEL
LIN {X 0,Y 474.681,Z 372.359,A -85,B 0,C 180,E1 -7315.56,E2 -7315.56} C_VEL
LIN {X 0,Y 474.652,Z 372.362,A -85,B 0,C 180,E1 -7318.283,E2 -7318.283} C_VEL
LIN {X 0,Y 474.604,Z 372.371,A -85,B 0,C 180,E1 -7321.218,E2 -7321.218} C_VEL
LIN {X 0,Y 474.638,Z 372.359,A -85,B 0,C 180,E1 -7324.242,E2 -7324.242} C_VEL
LIN {X 0,Y 474.596,Z 372.371,A -85,B 0,C 180,E1 -7327.384,E2 -7327.384} C_VEL
LIN {X 0,Y 474.633,Z 372.363,A -85,B 0,C 180,E1 -7329.648,E2 -7329.648} C_VEL
LIN {X 0,Y 474.637,Z 372.366,A -85,B 0,C 180,E1 -7332.933,E2 -7332.933} C_VEL
LIN {X 0,Y 474.615,Z 372.362,A -85,B 0,C 180,E1 -7335.896,E2 -7335.896} C_VEL
LIN {X 0,Y 474.633,Z 372.363,A -85,B 0,C 180,E1 -7339.041,E2 -7339.041} C_VEL
LIN {X 0,Y 474.615,Z 372.361,A -85,B 0,C 180,E1 -7341.704,E2 -7341.704} C_VEL
LIN {X 0,Y 474.63,Z 372.366,A -85,B 0,C 180,E1 -7344.726,E2 -7344.726} C_VEL
LIN {X 0,Y 474.641,Z 372.358,A -85,B 0,C 180,E1 -7347.788,E2 -7347.788} C_VEL
LIN {X 0,Y 474.629,Z 372.365,A -85,B 0,C 180,E1 -7350.885,E2 -7350.885} C_VEL
LIN {X 0,Y 474.659,Z 372.352,A -85,B 0,C 180,E1 -7353.628,E2 -7353.628} C_VEL
LIN {X 0,Y 474.64,Z 372.36,A -85,B 0,C 180,E1 -7356.642,E2 -7356.642} C_VEL
LIN {X 0,Y 474.66,Z 372.359,A -85,B 0,C 180,E1 -7360.09,E2 -7360.09} C_VEL
LIN {X 0,Y 474.654,Z 372.36,A -85,B 0,C 180,E1 -7362.775,E2 -7362.775} C_VEL
LIN {X 0,Y 474.653,Z 372.352,A -85,B 0,C 180,E1 -7365.421,E2 -7365.421} C_VEL
LIN {X 0,Y 474.71,Z 372.354,A -85,B 0,C 180,E1 -7368.038,E2 -7368.038} C_VEL
LIN {X 0,Y 474.733,Z 372.347,A -85,B 0,C 180,E1 -7371.487,E2 -7371.487} C_VEL
LIN {X 0,Y 474.785,Z 372.342,A -85,B 0,C 180,E1 -7374.053,E2 -7374.053} C_VEL
LIN {X 0,Y 474.9,Z 372.323,A -85,B 0,C 180,E1 -7377.455,E2 -7377.455} C_VEL
LIN {X 0,Y 474.917,Z 372.328,A -85,B 0,C 180,E1 -7380,E2 -7380} C_VEL
LIN {X 0,Y 474.9,Z 372.327,A -85,B 0,C 180,E1 -7382.545,E2 -7382.545} C_VEL
LIN {X 0,Y 474.785,Z 372.346,A -85,B 0,C 180,E1 -7385.948,E2 -7385.948} C_VEL
LIN {X 0,Y 474.734,Z 372.348,A -85,B 0,C 180,E1 -7388.514,E2 -7388.514} C_VEL
LIN {X 0,Y 474.71,Z 372.355,A -85,B 0,C 180,E1 -7391.962,E2 -7391.962} C_VEL
LIN {X 0,Y 474.706,Z 372.355,A -85,B 0,C 180,E1 -7395.456,E2 -7395.456} C_VEL
LIN {X 0,Y 474.671,Z 372.357,A -85,B 0,C 180,E1 -7399.01,E2 -7399.01} C_VEL
LIN {X 0,Y 474.595,Z 372.37,A -85,B 0,C 180,E1 -7401.729,E2 -7401.729} C_VEL
LIN {X 0,Y 474.647,Z 372.36,A -85,B 0,C 180,E1 -7404.494,E2 -7404.494} C_VEL
LIN {X 0,Y 474.687,Z 372.358,A -85,B 0,C 180,E1 -7407.334,E2 -7407.334} C_VEL
LIN {X 0,Y 474.661,Z 372.411,A -85,B 0,C 180,E1 -7410.104,E2 -7410.104} C_VEL
LIN {X 0,Y 476.031,Z 380.167,A -85,B 0,C 180,E1 -7411.857,E2 -7411.857} C_VEL
LIN {X 0,Y 475.609,Z 393.479,A -85,B 0,C 180,E1 -7414.674,E2 -7414.674} C_VEL
LIN {X 0,Y 475.473,Z 396.524,A -85,B 0,C 180,E1 -7415.302,E2 -7415.302} C_VEL
LIN {X 0,Y 478.224,Z 411.648,A -85,B 0,C 180,E1 -7415.645,E2 -7415.645} C_VEL
LIN {X 0,Y 477.397,Z 503.151,A -85,B 0,C 180,E1 -7417.073,E2 -7417.073} C_VEL
LIN {X 0,Y 477.107,Z 516.36,A -85,B 0,C 180,E1 -7417.447,E2 -7417.447} C_VEL
LIN {X 0,Y 476.768,Z 529.541,A -85,B 0,C 180,E1 -7418.007,E2 -7418.007} C_VEL
LIN {X 0,Y 476.366,Z 541.301,A -85,B 0,C 180,E1 -7418.691,E2 -7418.691} C_VEL
LIN {X 0,Y 475.846,Z 552.431,A -85,B 0,C 180,E1 -7419.52,E2 -7419.52} C_VEL
LIN {X 0,Y 475.388,Z 562.72,A -85,B 0,C 180,E1 -7420.476,E2 -7420.476} C_VEL
LIN {X 0,Y 474.95,Z 572.115,A -85,B 0,C 180,E1 -7421.557,E2 -7421.557} C_VEL
LIN {X 0,Y 474.577,Z 580.959,A -85,B 0,C 180,E1 -7422.821,E2 -7422.821} C_VEL
LIN {X 0,Y 474.26,Z 588.429,A -85,B 0,C 180,E1 -7424.146,E2 -7424.146} C_VEL
LIN {X 0,Y 474.058,Z 593.924,A -85,B 0,C 180,E1 -7425.366,E2 -7425.366} C_VEL
LIN {X 0,Y 473.892,Z 598.379,A -85,B 0,C 180,E1 -7426.61,E2 -7426.61} C_VEL
LIN {X 0,Y 473.783,Z 602.412,A -85,B 0,C 180,E1 -7428.123,E2 -7428.123} C_VEL
LIN {X 0,Y 473.648,Z 604.514,A -85,B 0,C 180,E1 -7429.24,E2 -7429.24} C_VEL
LIN {X 0,Y 473.606,Z 606.006,A -85,B 0,C 180,E1 -7430.502,E2 -7430.502} C_VEL
LIN {X 0,Y 473.601,Z 606.564,A -85,B 0,C 180,E1 -7431.447,E2 -7431.447} C_VEL
LIN {X 0,Y 472.926,Z 606.669,A -85,B 0,C 180,E1 -7432.158,E2 -7432.158} C_VEL
LIN {X 0,Y 470.07,Z 606.336,A -85,B 0,C 180,E1 -7433.312,E2 -7433.312} C_VEL
LIN {X 0,Y 467.678,Z 605.571,A -85,B 0,C 180,E1 -7434.237,E2 -7434.237} C_VEL
LIN {X 0,Y 466.67,Z 604.582,A -85,B 0,C 180,E1 -7434.944,E2 -7434.944} C_VEL
LIN {X 0,Y 466.599,Z 604.16,A -85,B 0,C 180,E1 -7435.181,E2 -7435.181} C_VEL
LIN {X 0,Y 466.735,Z 601.045,A -85,B 0,C 180,E1 -7436.659,E2 -7436.659} C_VEL
LIN {X 0,Y 466.926,Z 596.329,A -85,B 0,C 180,E1 -7438.209,E2 -7438.209} C_VEL
LIN {X 0,Y 467.141,Z 590.051,A -85,B 0,C 180,E1 -7439.734,E2 -7439.734} C_VEL
LIN {X 0,Y 467.445,Z 583.571,A -85,B 0,C 180,E1 -7440.977,E2 -7440.977} C_VEL
LIN {X 0,Y 467.831,Z 575.436,A -85,B 0,C 180,E1 -7442.244,E2 -7442.244} C_VEL
LIN {X 0,Y 468.242,Z 566.579,A -85,B 0,C 180,E1 -7443.358,E2 -7443.358} C_VEL
LIN {X 0,Y 468.802,Z 555.638,A -85,B 0,C 180,E1 -7444.468,E2 -7444.468} C_VEL
LIN {X 0,Y 469.247,Z 545.412,A -85,B 0,C 180,E1 -7445.302,E2 -7445.302} C_VEL
LIN {X 0,Y 469.671,Z 534.635,A -85,B 0,C 180,E1 -7446.004,E2 -7446.004} C_VEL
LIN {X 0,Y 470.024,Z 522.764,A -85,B 0,C 180,E1 -7446.597,E2 -7446.597} C_VEL
LIN {X 0,Y 470.382,Z 509.497,A -85,B 0,C 180,E1 -7447.067,E2 -7447.067} C_VEL
LIN {X 0,Y 470.573,Z 496.428,A -85,B 0,C 180,E1 -7447.351,E2 -7447.351} C_VEL
LIN {X 0,Y 471.274,Z 411.134,A -85,B 0,C 180,E1 -7448.682,E2 -7448.682} C_VEL
LIN {X 0,Y 468.457,Z 396.226,A -85,B 0,C 180,E1 -7449.039,E2 -7449.039} C_VEL
LIN {X 0,Y 469.038,Z 381.737,A -85,B 0,C 180,E1 -7452.11,E2 -7452.11} C_VEL
LIN {X 0,Y 467.697,Z 373.229,A -85,B 0,C 180,E1 -7454.049,E2 -7454.049} C_VEL
LIN {X 0,Y 467.662,Z 373.229,A -85,B 0,C 180,E1 -7457.854,E2 -7457.854} C_VEL
LIN {X 0,Y 467.687,Z 373.223,A -85,B 0,C 180,E1 -7461.356,E2 -7461.356} C_VEL
LIN {X 0,Y 467.726,Z 373.221,A -85,B 0,C 180,E1 -7463.961,E2 -7463.961} C_VEL
LIN {X 0,Y 467.864,Z 373.201,A -85,B 0,C 180,E1 -7467.416,E2 -7467.416} C_VEL
LIN {X 0,Y 467.887,Z 373.202,A -85,B 0,C 180,E1 -7469.999,E2 -7469.999} C_VEL
LIN {X 0,Y 467.863,Z 373.205,A -85,B 0,C 180,E1 -7472.582,E2 -7472.582} C_VEL
LIN {X 0,Y 467.746,Z 373.222,A -85,B 0,C 180,E1 -7476.036,E2 -7476.036} C_VEL
LIN {X 0,Y 467.683,Z 373.226,A -85,B 0,C 180,E1 -7478.642,E2 -7478.642} C_VEL
LIN {X 0,Y 467.658,Z 373.235,A -85,B 0,C 180,E1 -7482.144,E2 -7482.144} C_VEL
LIN {X 0,Y 467.668,Z 373.232,A -85,B 0,C 180,E1 -7485.892,E2 -7485.892} C_VEL
LIN {X 0,Y 467.624,Z 373.232,A -85,B 0,C 180,E1 -7489.306,E2 -7489.306} C_VEL
LIN {X 0,Y 467.534,Z 373.248,A -85,B 0,C 180,E1 -7492.072,E2 -7492.072} C_VEL
LIN {X 0,Y 467.583,Z 373.236,A -85,B 0,C 180,E1 -7494.887,E2 -7494.887} C_VEL
LIN {X 0,Y 467.626,Z 373.239,A -85,B 0,C 180,E1 -7497.767,E2 -7497.767} C_VEL
LIN {X 0,Y 467.57,Z 373.239,A -85,B 0,C 180,E1 -7501.045,E2 -7501.045} C_VEL
LIN {X 0,Y 467.587,Z 373.237,A -85,B 0,C 180,E1 -7504.241,E2 -7504.241} C_VEL
LIN {X 0,Y 467.548,Z 373.243,A -85,B 0,C 180,E1 -7507.186,E2 -7507.186} C_VEL
LIN {X 0,Y 467.592,Z 373.236,A -85,B 0,C 180,E1 -7510.261,E2 -7510.261} C_VEL
LIN {X 0,Y 467.581,Z 373.237,A -85,B 0,C 180,E1 -7512.566,E2 -7512.566} C_VEL
LIN {X 0,Y 467.565,Z 373.244,A -85,B 0,C 180,E1 -7515.052,E2 -7515.052} C_VEL
LIN {X 0,Y 467.604,Z 373.299,A -85,B 0,C 180,E1 -7516.724,E2 -7516.724} C_VEL
LIN {X 0,Y 468.681,Z 380.169,A -85,B 0,C 180,E1 -7518.111,E2 -7518.111} C_VEL
LIN {X 0,Y 468.35,Z 395.479,A -85,B 0,C 180,E1 -7521.079,E2 -7521.079} C_VEL
LIN {X 0,Y 471.197,Z 411.11,A -85,B 0,C 180,E1 -7521.461,E2 -7521.461} C_VEL
LIN {X 0,Y 470.263,Z 503.826,A -85,B 0,C 180,E1 -7522.987,E2 -7522.987} C_VEL
LIN {X 0,Y 469.982,Z 516.795,A -85,B 0,C 180,E1 -7523.368,E2 -7523.368} C_VEL
LIN {X 0,Y 469.624,Z 529.179,A -85,B 0,C 180,E1 -7523.91,E2 -7523.91} C_VEL
LIN {X 0,Y 469.179,Z 541.764,A -85,B 0,C 180,E1 -7524.649,E2 -7524.649} C_VEL
LIN {X 0,Y 468.748,Z 552.392,A -85,B 0,C 180,E1 -7525.456,E2 -7525.456} C_VEL
LIN {X 0,Y 468.236,Z 563.845,A -85,B 0,C 180,E1 -7526.549,E2 -7526.549} C_VEL
LIN {X 0,Y 467.823,Z 572.095,A -85,B 0,C 180,E1 -7527.516,E2 -7527.516} C_VEL
LIN {X 0,Y 467.534,Z 580.171,A -85,B 0,C 180,E1 -7528.662,E2 -7528.662} C_VEL
LIN {X 0,Y 467.158,Z 587.71,A -85,B 0,C 180,E1 -7529.985,E2 -7529.985} C_VEL
LIN {X 0,Y 466.983,Z 593.334,A -85,B 0,C 180,E1 -7531.21,E2 -7531.21} C_VEL
LIN {X 0,Y 466.783,Z 598.573,A -85,B 0,C 180,E1 -7532.659,E2 -7532.659} C_VEL
LIN {X 0,Y 466.662,Z 602.408,A -85,B 0,C 180,E1 -7534.103,E2 -7534.103} C_VEL
LIN {X 0,Y 466.573,Z 604.226,A -85,B 0,C 180,E1 -7535.054,E2 -7535.054} C_VEL
LIN {X 0,Y 466.515,Z 605.57,A -85,B 0,C 180,E1 -7535.999,E2 -7535.999} C_VEL
LIN {X 0,Y 466.528,Z 606.371,A -85,B 0,C 180,E1 -7536.941,E2 -7536.941} C_VEL
LIN {X 0,Y 466.495,Z 606.715,A -85,B 0,C 180,E1 -7537.874,E2 -7537.874} C_VEL
LIN {X 0,Y 466.534,Z 606.453,A -85,B 0,C 180,E1 -7539.06,E2 -7539.06} C_VEL
LIN {X 0,Y 466.58,Z 604.925,A -85,B 0,C 180,E1 -7540.647,E2 -7540.647} C_VEL
LIN {X 0,Y 466.634,Z 603.334,A -85,B 0,C 180,E1 -7541.589,E2 -7541.589} C_VEL
LIN {X 0,Y 466.746,Z 600.199,A -85,B 0,C 180,E1 -7542.925,E2 -7542.925} C_VEL
LIN {X 0,Y 466.876,Z 595.258,A -85,B 0,C 180,E1 -7544.446,E2 -7544.446} C_VEL
LIN {X 0,Y 467.174,Z 589.236,A -85,B 0,C 180,E1 -7545.85,E2 -7545.85} C_VEL
LIN {X 0,Y 467.427,Z 581.914,A -85,B 0,C 180,E1 -7547.193,E2 -7547.193} C_VEL
LIN {X 0,Y 467.872,Z 572.888,A -85,B 0,C 180,E1 -7548.52,E2 -7548.52} C_VEL
LIN {X 0,Y 468.304,Z 563.477,A -85,B 0,C 180,E1 -7549.625,E2 -7549.625} C_VEL
LIN {X 0,Y 468.786,Z 553.077,A -85,B 0,C 180,E1 -7550.617,E2 -7550.617} C_VEL
LIN {X 0,Y 469.262,Z 542.244,A -85,B 0,C 180,E1 -7551.447,E2 -7551.447} C_VEL
LIN {X 0,Y 469.721,Z 530.221,A -85,B 0,C 180,E1 -7552.16,E2 -7552.16} C_VEL
LIN {X 0,Y 470.03,Z 518.244,A -85,B 0,C 180,E1 -7552.698,E2 -7552.698} C_VEL
LIN {X 0,Y 470.308,Z 506.096,A -85,B 0,C 180,E1 -7553.08,E2 -7553.08} C_VEL
LIN {X 0,Y 470.57,Z 484.729,A -85,B 0,C 180,E1 -7553.461,E2 -7553.461} C_VEL
LIN {X 0,Y 471.311,Z 410.76,A -85,B 0,C 180,E1 -7554.693,E2 -7554.693} C_VEL
LIN {X 0,Y 468.444,Z 395.998,A -85,B 0,C 180,E1 -7555.078,E2 -7555.078} C_VEL
LIN {X 0,Y 468.739,Z 380.259,A -85,B 0,C 180,E1 -7558.067,E2 -7558.067} C_VEL
LIN {X 0,Y 467.846,Z 373.211,A -85,B 0,C 180,E1 -7559.462,E2 -7559.462} C_VEL
LIN {X 0,Y 467.851,Z 373.212,A -85,B 0,C 180,E1 -7562.583,E2 -7562.583} C_VEL
LIN {X 0,Y 467.734,Z 373.225,A -85,B 0,C 180,E1 -7566.037,E2 -7566.037} C_VEL
LIN {X 0,Y 467.672,Z 373.232,A -85,B 0,C 180,E1 -7568.643,E2 -7568.643} C_VEL
LIN {X 0,Y 467.672,Z 373.231,A -85,B 0,C 180,E1 -7572.145,E2 -7572.145} C_VEL
LIN {X 0,Y 467.656,Z 373.234,A -85,B 0,C 180,E1 -7575.893,E2 -7575.893} C_VEL
LIN {X 0,Y 467.614,Z 373.235,A -85,B 0,C 180,E1 -7579.308,E2 -7579.308} C_VEL
LIN {X 0,Y 467.568,Z 373.245,A -85,B 0,C 180,E1 -7582.072,E2 -7582.072} C_VEL
LIN {X 0,Y 467.608,Z 373.234,A -85,B 0,C 180,E1 -7584.887,E2 -7584.887} C_VEL
LIN {X 0,Y 467.619,Z 373.239,A -85,B 0,C 180,E1 -7587.769,E2 -7587.769} C_VEL
LIN {X 0,Y 467.564,Z 373.242,A -85,B 0,C 180,E1 -7591.047,E2 -7591.047} C_VEL
LIN {X 0,Y 467.581,Z 373.239,A -85,B 0,C 180,E1 -7594.244,E2 -7594.244} C_VEL
LIN {X 0,Y 467.542,Z 373.247,A -85,B 0,C 180,E1 -7597.188,E2 -7597.188} C_VEL
LIN {X 0,Y 467.571,Z 373.239,A -85,B 0,C 180,E1 -7600.265,E2 -7600.265} C_VEL
LIN {X 0,Y 467.579,Z 373.238,A -85,B 0,C 180,E1 -7602.568,E2 -7602.568} C_VEL
LIN {X 0,Y 467.564,Z 373.245,A -85,B 0,C 180,E1 -7605.054,E2 -7605.054} C_VEL
LIN {X 0,Y 467.582,Z 373.242,A -85,B 0,C 180,E1 -7607.441,E2 -7607.441} C_VEL
LIN {X 0,Y 467.577,Z 373.243,A -85,B 0,C 180,E1 -7610.857,E2 -7610.857} C_VEL
LIN {X 0,Y 467.559,Z 373.241,A -85,B 0,C 180,E1 -7614.261,E2 -7614.261} C_VEL
LIN {X 0,Y 467.578,Z 373.241,A -85,B 0,C 180,E1 -7617.322,E2 -7617.322} C_VEL
LIN {X 0,Y 467.576,Z 373.244,A -85,B 0,C 180,E1 -7620.667,E2 -7620.667} C_VEL
LIN {X 0,Y 467.626,Z 373.238,A -85,B 0,C 180,E1 -7623.202,E2 -7623.202} C_VEL
LIN {X 0,Y 467.662,Z 373.434,A -85,B 0,C 180,E1 -7624.282,E2 -7624.282} C_VEL
LIN {X 0,Y 469.876,Z 385.513,A -85,B 0,C 180,E1 -7626.65,E2 -7626.65} C_VEL
LIN {X 0,Y 469.246,Z 399.393,A -85,B 0,C 180,E1 -7629.164,E2 -7629.164} C_VEL
LIN {X 0,Y 468.622,Z 414.52,A -85,B 0,C 180,E1 -7631.87,E2 -7631.87} C_VEL
LIN {X 0,Y 468.357,Z 420.817,A -85,B 0,C 180,E1 -7632.987,E2 -7632.987} C_VEL
LIN {X 0,Y 471.21,Z 439.321,A -85,B 0,C 180,E1 -7633.397,E2 -7633.397} C_VEL
LIN {X 0,Y 470.468,Z 529.22,A -85,B 0,C 180,E1 -7634.819,E2 -7634.819} C_VEL
LIN {X 0,Y 470.108,Z 542.357,A -85,B 0,C 180,E1 -7635.195,E2 -7635.195} C_VEL
LIN {X 0,Y 469.709,Z 554.472,A -85,B 0,C 180,E1 -7635.708,E2 -7635.708} C_VEL
LIN {X 0,Y 469.244,Z 565.91,A -85,B 0,C 180,E1 -7636.357,E2 -7636.357} C_VEL
LIN {X 0,Y 468.673,Z 577.923,A -85,B 0,C 180,E1 -7637.245,E2 -7637.245} C_VEL
LIN {X 0,Y 468.258,Z 588.226,A -85,B 0,C 180,E1 -7638.201,E2 -7638.201} C_VEL
LIN {X 0,Y 467.806,Z 596.855,A -85,B 0,C 180,E1 -7639.177,E2 -7639.177} C_VEL
LIN {X 0,Y 467.45,Z 604.811,A -85,B 0,C 180,E1 -7640.263,E2 -7640.263} C_VEL
LIN {X 0,Y 467.116,Z 612.586,A -85,B 0,C 180,E1 -7641.566,E2 -7641.566} C_VEL
LIN {X 0,Y 466.853,Z 619.73,A -85,B 0,C 180,E1 -7643.084,E2 -7643.084} C_VEL
LIN {X 0,Y 466.767,Z 624.487,A -85,B 0,C 180,E1 -7644.385,E2 -7644.385} C_VEL
LIN {X 0,Y 466.646,Z 628.119,A -85,B 0,C 180,E1 -7645.683,E2 -7645.683} C_VEL
LIN {X 0,Y 466.688,Z 629.994,A -85,B 0,C 180,E1 -7646.548,E2 -7646.548} C_VEL
LIN {X 0,Y 466.661,Z 631.398,A -85,B 0,C 180,E1 -7647.412,E2 -7647.412} C_VEL
LIN {X 0,Y 466.618,Z 633.004,A -85,B 0,C 180,E1 -7649.138,E2 -7649.138} C_VEL
LIN {X 0,Y 466.598,Z 633.218,A -85,B 0,C 180,E1 -7650.001,E2 -7650.001} C_VEL
LIN {X 0,Y 466.618,Z 632.996,A -85,B 0,C 180,E1 -7650.864,E2 -7650.864} C_VEL
LIN {X 0,Y 466.662,Z 631.372,A -85,B 0,C 180,E1 -7652.591,E2 -7652.591} C_VEL
LIN {X 0,Y 466.689,Z 629.96,A -85,B 0,C 180,E1 -7653.455,E2 -7653.455} C_VEL
LIN {X 0,Y 466.691,Z 626.995,A -85,B 0,C 180,E1 -7654.752,E2 -7654.752} C_VEL
LIN {X 0,Y 466.759,Z 622.984,A -85,B 0,C 180,E1 -7656.051,E2 -7656.051} C_VEL
LIN {X 0,Y 466.951,Z 616.815,A -85,B 0,C 180,E1 -7657.569,E2 -7657.569} C_VEL
LIN {X 0,Y 467.227,Z 610.08,A -85,B 0,C 180,E1 -7658.87,E2 -7658.87} C_VEL
LIN {X 0,Y 467.562,Z 601.725,A -85,B 0,C 180,E1 -7660.174,E2 -7660.174} C_VEL
LIN {X 0,Y 468.008,Z 593.143,A -85,B 0,C 180,E1 -7661.259,E2 -7661.259} C_VEL
LIN {X 0,Y 468.509,Z 583.009,A -85,B 0,C 180,E1 -7662.301,E2 -7662.301} C_VEL
LIN {X 0,Y 468.934,Z 572.066,A -85,B 0,C 180,E1 -7663.213,E2 -7663.213} C_VEL
LIN {X 0,Y 469.455,Z 560.544,A -85,B 0,C 180,E1 -7663.97,E2 -7663.97} C_VEL
LIN {X 0,Y 469.919,Z 548.615,A -85,B 0,C 180,E1 -7664.564,E2 -7664.564} C_VEL
LIN {X 0,Y 470.275,Z 535.769,A -85,B 0,C 180,E1 -7665.023,E2 -7665.023} C_VEL
LIN {X 0,Y 470.614,Z 522.371,A -85,B 0,C 180,E1 -7665.317,E2 -7665.317} C_VEL
LIN {X 0,Y 471.118,Z 437.973,A -85,B 0,C 180,E1 -7666.645,E2 -7666.645} C_VEL
LIN {X 0,Y 468.305,Z 420.511,A -85,B 0,C 180,E1 -7667.035,E2 -7667.035} C_VEL
LIN {X 0,Y 468.942,Z 405.503,A -85,B 0,C 180,E1 -7669.708,E2 -7669.708} C_VEL
LIN {X 0,Y 469.753,Z 389.173,A -85,B 0,C 180,E1 -7672.66,E2 -7672.66} C_VEL
LIN {X 0,Y 469.759,Z 384.158,A -85,B 0,C 180,E1 -7673.592,E2 -7673.592} C_VEL
LIN {X 0,Y 467.64,Z 373.237,A -85,B 0,C 180,E1 -7675.799,E2 -7675.799} C_VEL
LIN {X 0,Y 467.583,Z 373.244,A -85,B 0,C 180,E1 -7678.75,E2 -7678.75} C_VEL
LIN {X 0,Y 467.588,Z 373.242,A -85,B 0,C 180,E1 -7681.741,E2 -7681.741} C_VEL
LIN {X 0,Y 467.571,Z 373.243,A -85,B 0,C 180,E1 -7684.833,E2 -7684.833} C_VEL
LIN {X 0,Y 467.571,Z 373.242,A -85,B 0,C 180,E1 -7688.045,E2 -7688.045} C_VEL
LIN {X 0,Y 467.583,Z 373.245,A -85,B 0,C 180,E1 -7691.277,E2 -7691.277} C_VEL
LIN {X 0,Y 467.56,Z 373.242,A -85,B 0,C 180,E1 -7693.821,E2 -7693.821} C_VEL
LIN {X 0,Y 467.562,Z 373.242,A -85,B 0,C 180,E1 -7696.256,E2 -7696.256} C_VEL
LIN {X 0,Y 467.583,Z 373.243,A -85,B 0,C 180,E1 -7698.724,E2 -7698.724} C_VEL
LIN {X 0,Y 467.57,Z 373.239,A -85,B 0,C 180,E1 -7701.956,E2 -7701.956} C_VEL
LIN {X 0,Y 467.569,Z 373.24,A -85,B 0,C 180,E1 -7705.168,E2 -7705.168} C_VEL
LIN {X 0,Y 467.588,Z 373.239,A -85,B 0,C 180,E1 -7708.26,E2 -7708.26} C_VEL
LIN {X 0,Y 467.581,Z 373.239,A -85,B 0,C 180,E1 -7711.251,E2 -7711.251} C_VEL
LIN {X 0,Y 467.602,Z 373.234,A -85,B 0,C 180,E1 -7714.16,E2 -7714.16} C_VEL
LIN {X 0,Y 467.581,Z 373.236,A -85,B 0,C 180,E1 -7716.996,E2 -7716.996} C_VEL
LIN {X 0,Y 467.628,Z 373.232,A -85,B 0,C 180,E1 -7719.777,E2 -7719.777} C_VEL
LIN {X 0,Y 467.613,Z 373.239,A -85,B 0,C 180,E1 -7722.507,E2 -7722.507} C_VEL
LIN {X 0,Y 467.611,Z 373.229,A -85,B 0,C 180,E1 -7725.197,E2 -7725.197} C_VEL
LIN {X 0,Y 467.662,Z 373.23,A -85,B 0,C 180,E1 -7727.855,E2 -7727.855} C_VEL
LIN {X 0,Y 467.687,Z 373.224,A -85,B 0,C 180,E1 -7731.357,E2 -7731.357} C_VEL
LIN {X 0,Y 467.749,Z 373.217,A -85,B 0,C 180,E1 -7733.963,E2 -7733.963} C_VEL
LIN {X 0,Y 467.865,Z 373.199,A -85,B 0,C 180,E1 -7737.417,E2 -7737.417} C_VEL
LIN {X 0,Y 467.888,Z 373.204,A -85,B 0,C 180,E1 -7740,E2 -7740} C_VEL
LIN {X 0,Y 467.865,Z 373.203,A -85,B 0,C 180,E1 -7742.583,E2 -7742.583} C_VEL
LIN {X 0,Y 467.749,Z 373.221,A -85,B 0,C 180,E1 -7746.037,E2 -7746.037} C_VEL
LIN {X 0,Y 467.687,Z 373.225,A -85,B 0,C 180,E1 -7748.643,E2 -7748.643} C_VEL
LIN {X 0,Y 467.662,Z 373.232,A -85,B 0,C 180,E1 -7752.145,E2 -7752.145} C_VEL
LIN {X 0,Y 467.645,Z 373.236,A -85,B 0,C 180,E1 -7755.695,E2 -7755.695} C_VEL
LIN {X 0,Y 467.623,Z 373.234,A -85,B 0,C 180,E1 -7758.764,E2 -7758.764} C_VEL
LIN {X 0,Y 467.587,Z 373.241,A -85,B 0,C 180,E1 -7761.268,E2 -7761.268} C_VEL
LIN {X 0,Y 467.569,Z 373.244,A -85,B 0,C 180,E1 -7763.944,E2 -7763.944} C_VEL
LIN {X 0,Y 467.619,Z 373.237,A -85,B 0,C 180,E1 -7766.8,E2 -7766.8} C_VEL
LIN {X 0,Y 467.663,Z 373.375,A -85,B 0,C 180,E1 -7769.917,E2 -7769.917} C_VEL
LIN {X 0,Y 469.112,Z 381.923,A -85,B 0,C 180,E1 -7771.877,E2 -7771.877} C_VEL
LIN {X 0,Y 468.605,Z 395.292,A -85,B 0,C 180,E1 -7774.744,E2 -7774.744} C_VEL
LIN {X 0,Y 468.551,Z 396.866,A -85,B 0,C 180,E1 -7775.044,E2 -7775.044} C_VEL
LIN {X 0,Y 471.409,Z 411.388,A -85,B 0,C 180,E1 -7775.388,E2 -7775.388} C_VEL
LIN {X 0,Y 470.559,Z 503.551,A -85,B 0,C 180,E1 -7776.852,E2 -7776.852} C_VEL
LIN {X 0,Y 470.256,Z 516.695,A -85,B 0,C 180,E1 -7777.232,E2 -7777.232} C_VEL
LIN {X 0,Y 469.919,Z 528.676,A -85,B 0,C 180,E1 -7777.743,E2 -7777.743} C_VEL
LIN {X 0,Y 469.509,Z 540.251,A -85,B 0,C 180,E1 -7778.405,E2 -7778.405} C_VEL
LIN {X 0,Y 468.98,Z 552.05,A -85,B 0,C 180,E1 -7779.283,E2 -7779.283} C_VEL
LIN {X 0,Y 468.438,Z 563.063,A -85,B 0,C 180,E1 -7780.317,E2 -7780.317} C_VEL
LIN {X 0,Y 467.989,Z 572.012,A -85,B 0,C 180,E1 -7781.359,E2 -7781.359} C_VEL
LIN {X 0,Y 467.626,Z 580.471,A -85,B 0,C 180,E1 -7782.571,E2 -7782.571} C_VEL
LIN {X 0,Y 467.249,Z 587.377,A -85,B 0,C 180,E1 -7783.781,E2 -7783.781} C_VEL
LIN {X 0,Y 466.989,Z 593.11,A -85,B 0,C 180,E1 -7785.019,E2 -7785.019} C_VEL
LIN {X 0,Y 466.843,Z 597.744,A -85,B 0,C 180,E1 -7786.27,E2 -7786.27} C_VEL
LIN {X 0,Y 466.729,Z 601.411,A -85,B 0,C 180,E1 -7787.548,E2 -7787.548} C_VEL
LIN {X 0,Y 466.598,Z 604.156,A -85,B 0,C 180,E1 -7788.861,E2 -7788.861} C_VEL
LIN {X 0,Y 466.53,Z 605.954,A -85,B 0,C 180,E1 -7790.201,E2 -7790.201} C_VEL
LIN {X 0,Y 466.508,Z 606.839,A -85,B 0,C 180,E1 -7791.853,E2 -7791.853} C_VEL
LIN {X 0,Y 466.521,Z 606.602,A -85,B 0,C 180,E1 -7792.981,E2 -7792.981} C_VEL
LIN {X 0,Y 466.551,Z 605.296,A -85,B 0,C 180,E1 -7794.434,E2 -7794.434} C_VEL
LIN {X 0,Y 466.599,Z 604.16,A -85,B 0,C 180,E1 -7795.181,E2 -7795.181} C_VEL
LIN {X 0,Y 465.978,Z 602.894,A -85,B 0,C 180,E1 -7795.882,E2 -7795.882} C_VEL
LIN {X 0,Y 463.225,Z 600.299,A -85,B 0,C 180,E1 -7797.012,E2 -7797.012} C_VEL
LIN {X 0,Y 460.915,Z 597.753,A -85,B 0,C 180,E1 -7797.907,E2 -7797.907} C_VEL
LIN {X 0,Y 459.971,Z 595.486,A -85,B 0,C 180,E1 -7798.582,E2 -7798.582} C_VEL
LIN {X 0,Y 459.92,Z 594.656,A -85,B 0,C 180,E1 -7798.807,E2 -7798.807} C_VEL
LIN {X 0,Y 460.171,Z 588.836,A -85,B 0,C 180,E1 -7800.149,E2 -7800.149} C_VEL
LIN {X 0,Y 460.512,Z 581.363,A -85,B 0,C 180,E1 -7801.515,E2 -7801.515} C_VEL
LIN {X 0,Y 460.946,Z 572.781,A -85,B 0,C 180,E1 -7802.779,E2 -7802.779} C_VEL
LIN {X 0,Y 461.409,Z 564.43,A -85,B 0,C 180,E1 -7803.786,E2 -7803.786} C_VEL
LIN {X 0,Y 461.93,Z 554.339,A -85,B 0,C 180,E1 -7804.785,E2 -7804.785} C_VEL
LIN {X 0,Y 462.403,Z 543.225,A -85,B 0,C 180,E1 -7805.664,E2 -7805.664} C_VEL
LIN {X 0,Y 462.908,Z 531.43,A -85,B 0,C 180,E1 -7806.394,E2 -7806.394} C_VEL
LIN {X 0,Y 463.264,Z 519.798,A -85,B 0,C 180,E1 -7806.94,E2 -7806.94} C_VEL
LIN {X 0,Y 463.6,Z 506.93,A -85,B 0,C 180,E1 -7807.358,E2 -7807.358} C_VEL
LIN {X 0,Y 463.792,Z 489.724,A -85,B 0,C 180,E1 -7807.68,E2 -7807.68} C_VEL
LIN {X 0,Y 464.509,Z 412.233,A -85,B 0,C 180,E1 -7808.911,E2 -7808.911} C_VEL
LIN {X 0,Y 461.52,Z 396.418,A -85,B 0,C 180,E1 -7809.293,E2 -7809.293} C_VEL
LIN {X 0,Y 462.052,Z 382.493,A -85,B 0,C 180,E1 -7812.288,E2 -7812.288} C_VEL
LIN {X 0,Y 460.647,Z 374.107,A -85,B 0,C 180,E1 -7814.245,E2 -7814.245} C_VEL
LIN {X 0,Y 460.615,Z 374.107,A -85,B 0,C 180,E1 -7817.665,E2 -7817.665} C_VEL
LIN {X 0,Y 460.634,Z 374.103,A -85,B 0,C 180,E1 -7821.223,E2 -7821.223} C_VEL
LIN {X 0,Y 460.69,Z 374.096,A -85,B 0,C 180,E1 -7823.869,E2 -7823.869} C_VEL
LIN {X 0,Y 460.805,Z 374.081,A -85,B 0,C 180,E1 -7827.376,E2 -7827.376} C_VEL
LIN {X 0,Y 460.857,Z 374.078,A -85,B 0,C 180,E1 -7829.999,E2 -7829.999} C_VEL
LIN {X 0,Y 460.828,Z 374.081,A -85,B 0,C 180,E1 -7832.621,E2 -7832.621} C_VEL
LIN {X 0,Y 460.713,Z 374.099,A -85,B 0,C 180,E1 -7836.129,E2 -7836.129} C_VEL
LIN {X 0,Y 460.63,Z 374.104,A -85,B 0,C 180,E1 -7838.775,E2 -7838.775} C_VEL
LIN {X 0,Y 460.615,Z 374.108,A -85,B 0,C 180,E1 -7842.444,E2 -7842.444} C_VEL
LIN {X 0,Y 460.623,Z 374.111,A -85,B 0,C 180,E1 -7846.006,E2 -7846.006} C_VEL
LIN {X 0,Y 460.569,Z 374.114,A -85,B 0,C 180,E1 -7849.614,E2 -7849.614} C_VEL
LIN {X 0,Y 460.51,Z 374.119,A -85,B 0,C 180,E1 -7852.427,E2 -7852.427} C_VEL
LIN {X 0,Y 460.551,Z 374.12,A -85,B 0,C 180,E1 -7855.797,E2 -7855.797} C_VEL
LIN {X 0,Y 460.556,Z 374.114,A -85,B 0,C 180,E1 -7858.231,E2 -7858.231} C_VEL
LIN {X 0,Y 460.522,Z 374.118,A -85,B 0,C 180,E1 -7861.283,E2 -7861.283} C_VEL
LIN {X 0,Y 460.531,Z 374.115,A -85,B 0,C 180,E1 -7864.505,E2 -7864.505} C_VEL
LIN {X 0,Y 460.527,Z 374.123,A -85,B 0,C 180,E1 -7867.619,E2 -7867.619} C_VEL
LIN {X 0,Y 460.554,Z 374.112,A -85,B 0,C 180,E1 -7870.271,E2 -7870.271} C_VEL
LIN {X 0,Y 460.503,Z 374.125,A -85,B 0,C 180,E1 -7873.373,E2 -7873.373} C_VEL
LIN {X 0,Y 460.578,Z 374.225,A -85,B 0,C 180,E1 -7876.6,E2 -7876.6} C_VEL
LIN {X 0,Y 461.69,Z 380.856,A -85,B 0,C 180,E1 -7877.949,E2 -7877.949} C_VEL
LIN {X 0,Y 461.384,Z 395.683,A -85,B 0,C 180,E1 -7880.846,E2 -7880.846} C_VEL
LIN {X 0,Y 464.343,Z 411.9,A -85,B 0,C 180,E1 -7881.233,E2 -7881.233} C_VEL
LIN {X 0,Y 463.361,Z 504.026,A -85,B 0,C 180,E1 -7882.784,E2 -7882.784} C_VEL
LIN {X 0,Y 463.092,Z 516.804,A -85,B 0,C 180,E1 -7883.165,E2 -7883.165} C_VEL
LIN {X 0,Y 462.688,Z 529.72,A -85,B 0,C 180,E1 -7883.74,E2 -7883.74} C_VEL
LIN {X 0,Y 462.261,Z 541.483,A -85,B 0,C 180,E1 -7884.441,E2 -7884.441} C_VEL
LIN {X 0,Y 461.796,Z 552.288,A -85,B 0,C 180,E1 -7885.264,E2 -7885.264} C_VEL
LIN {X 0,Y 461.276,Z 563.519,A -85,B 0,C 180,E1 -7886.343,E2 -7886.343} C_VEL
LIN {X 0,Y 460.786,Z 573.14,A -85,B 0,C 180,E1 -7887.49,E2 -7887.49} C_VEL
LIN {X 0,Y 460.452,Z 581.555,A -85,B 0,C 180,E1 -7888.738,E2 -7888.738} C_VEL
LIN {X 0,Y 460.038,Z 589.382,A -85,B 0,C 180,E1 -7890.178,E2 -7890.178} C_VEL
LIN {X 0,Y 459.814,Z 595.807,A -85,B 0,C 180,E1 -7891.717,E2 -7891.717} C_VEL
LIN {X 0,Y 459.653,Z 600.468,A -85,B 0,C 180,E1 -7893.189,E2 -7893.189} C_VEL
LIN {X 0,Y 459.526,Z 603.781,A -85,B 0,C 180,E1 -7894.644,E2 -7894.644} C_VEL
LIN {X 0,Y 459.438,Z 605.278,A -85,B 0,C 180,E1 -7895.605,E2 -7895.605} C_VEL
LIN {X 0,Y 459.434,Z 606.346,A -85,B 0,C 180,E1 -7896.606,E2 -7896.606} C_VEL
LIN {X 0,Y 459.4,Z 606.831,A -85,B 0,C 180,E1 -7897.514,E2 -7897.514} C_VEL
LIN {X 0,Y 459.444,Z 606.729,A -85,B 0,C 180,E1 -7898.919,E2 -7898.919} C_VEL
LIN {X 0,Y 459.488,Z 605.564,A -85,B 0,C 180,E1 -7900.336,E2 -7900.336} C_VEL
LIN {X 0,Y 459.549,Z 603.88,A -85,B 0,C 180,E1 -7901.469,E2 -7901.469} C_VEL
LIN {X 0,Y 459.675,Z 600.093,A -85,B 0,C 180,E1 -7903.112,E2 -7903.112} C_VEL
LIN {X 0,Y 459.838,Z 595.086,A -85,B 0,C 180,E1 -7904.651,E2 -7904.651} C_VEL
LIN {X 0,Y 460.152,Z 588.901,A -85,B 0,C 180,E1 -7906.081,E2 -7906.081} C_VEL
LIN {X 0,Y 460.465,Z 581.355,A -85,B 0,C 180,E1 -7907.461,E2 -7907.461} C_VEL
LIN {X 0,Y 460.851,Z 573.924,A -85,B 0,C 180,E1 -7908.565,E2 -7908.565} C_VEL
LIN {X 0,Y 461.283,Z 564.751,A -85,B 0,C 180,E1 -7909.687,E2 -7909.687} C_VEL
LIN {X 0,Y 461.777,Z 554.557,A -85,B 0,C 180,E1 -7910.694,E2 -7910.694} C_VEL
LIN {X 0,Y 462.35,Z 542.875,A -85,B 0,C 180,E1 -7911.618,E2 -7911.618} C_VEL
LIN {X 0,Y 462.808,Z 531.615,A -85,B 0,C 180,E1 -7912.309,E2 -7912.309} C_VEL
LIN {X 0,Y 463.178,Z 518.426,A -85,B 0,C 180,E1 -7912.918,E2 -7912.918} C_VEL
LIN {X 0,Y 463.473,Z 506.273,A -85,B 0,C 180,E1 -7913.306,E2 -7913.306} C_VEL
LIN {X 0,Y 463.766,Z 481.939,A -85,B 0,C 180,E1 -7913.747,E2 -7913.747} C_VEL
LIN {X 0,Y 464.497,Z 411.362,A -85,B 0,C 180,E1 -7914.954,E2 -7914.954} C_VEL
LIN {X 0,Y 461.542,Z 396.178,A -85,B 0,C 180,E1 -7915.36,E2 -7915.36} C_VEL
LIN {X 0,Y 461.787,Z 382.118,A -85,B 0,C 180,E1 -7918.038,E2 -7918.038} C_VEL
LIN {X 0,Y 460.824,Z 374.086,A -85,B 0,C 180,E1 -7919.618,E2 -7919.618} C_VEL
LIN {X 0,Y 460.816,Z 374.088,A -85,B 0,C 180,E1 -7922.622,E2 -7922.622} C_VEL
LIN {X 0,Y 460.7,Z 374.102,A -85,B 0,C 180,E1 -7926.13,E2 -7926.13} C_VEL
LIN {X 0,Y 460.619,Z 374.109,A -85,B 0,C 180,E1 -7928.776,E2 -7928.776} C_VEL
LIN {X 0,Y 460.623,Z 374.109,A -85,B 0,C 180,E1 -7932.457,E2 -7932.457} C_VEL
LIN {X 0,Y 460.611,Z 374.113,A -85,B 0,C 180,E1 -7936.008,E2 -7936.008} C_VEL
LIN {X 0,Y 460.56,Z 374.116,A -85,B 0,C 180,E1 -7939.616,E2 -7939.616} C_VEL
LIN {X 0,Y 460.531,Z 374.117,A -85,B 0,C 180,E1 -7942.428,E2 -7942.428} C_VEL
LIN {X 0,Y 460.576,Z 374.116,A -85,B 0,C 180,E1 -7945.807,E2 -7945.807} C_VEL
LIN {X 0,Y 460.549,Z 374.117,A -85,B 0,C 180,E1 -7948.233,E2 -7948.233} C_VEL
LIN {X 0,Y 460.516,Z 374.122,A -85,B 0,C 180,E1 -7951.285,E2 -7951.285} C_VEL
LIN {X 0,Y 460.525,Z 374.117,A -85,B 0,C 180,E1 -7954.507,E2 -7954.507} C_VEL
LIN {X 0,Y 460.52,Z 374.123,A -85,B 0,C 180,E1 -7957.621,E2 -7957.621} C_VEL
LIN {X 0,Y 460.535,Z 374.116,A -85,B 0,C 180,E1 -7960.271,E2 -7960.271} C_VEL
LIN {X 0,Y 460.502,Z 374.126,A -85,B 0,C 180,E1 -7963.375,E2 -7963.375} C_VEL
LIN {X 0,Y 460.503,Z 374.121,A -85,B 0,C 180,E1 -7966.627,E2 -7966.627} C_VEL
LIN {X 0,Y 460.537,Z 374.117,A -85,B 0,C 180,E1 -7969.732,E2 -7969.732} C_VEL
LIN {X 0,Y 460.522,Z 374.119,A -85,B 0,C 180,E1 -7972.52,E2 -7972.52} C_VEL
LIN {X 0,Y 460.544,Z 374.116,A -85,B 0,C 180,E1 -7975.625,E2 -7975.625} C_VEL
LIN {X 0,Y 460.533,Z 374.122,A -85,B 0,C 180,E1 -7978.746,E2 -7978.746} C_VEL
LIN {X 0,Y 460.556,Z 374.115,A -85,B 0,C 180,E1 -7981.769,E2 -7981.769} C_VEL
LIN {X 0,Y 460.611,Z 374.199,A -85,B 0,C 180,E1 -7984.046,E2 -7984.046} C_VEL
LIN {X 0,Y 462.909,Z 386.569,A -85,B 0,C 180,E1 -7986.515,E2 -7986.515} C_VEL
LIN {X 0,Y 462.279,Z 400.454,A -85,B 0,C 180,E1 -7989.069,E2 -7989.069} C_VEL
LIN {X 0,Y 461.605,Z 415.576,A -85,B 0,C 180,E1 -7991.815,E2 -7991.815} C_VEL
LIN {X 0,Y 461.39,Z 420.831,A -85,B 0,C 180,E1 -7992.744,E2 -7992.744} C_VEL
LIN {X 0,Y 464.418,Z 439.984,A -85,B 0,C 180,E1 -7993.167,E2 -7993.167} C_VEL
LIN {X 0,Y 463.634,Z 528.634,A -85,B 0,C 180,E1 -7994.59,E2 -7994.59} C_VEL
LIN {X 0,Y 463.208,Z 541.898,A -85,B 0,C 180,E1 -7994.97,E2 -7994.97} C_VEL
LIN {X 0,Y 462.789,Z 554.083,A -85,B 0,C 180,E1 -7995.49,E2 -7995.49} C_VEL
LIN {X 0,Y 462.311,Z 565.575,A -85,B 0,C 180,E1 -7996.148,E2 -7996.148} C_VEL
LIN {X 0,Y 461.735,Z 577.629,A -85,B 0,C 180,E1 -7997.05,E2 -7997.05} C_VEL
LIN {X 0,Y 461.284,Z 587.955,A -85,B 0,C 180,E1 -7998.02,E2 -7998.02} C_VEL
LIN {X 0,Y 460.807,Z 596.599,A -85,B 0,C 180,E1 -7999.011,E2 -7999.011} C_VEL
LIN {X 0,Y 460.422,Z 604.566,A -85,B 0,C 180,E1 -8000.113,E2 -8000.113} C_VEL
LIN {X 0,Y 460.052,Z 612.354,A -85,B 0,C 180,E1 -8001.435,E2 -8001.435} C_VEL
LIN {X 0,Y 459.773,Z 619.506,A -85,B 0,C 180,E1 -8002.977,E2 -8002.977} C_VEL
LIN {X 0,Y 459.664,Z 624.27,A -85,B 0,C 180,E1 -8004.298,E2 -8004.298} C_VEL
LIN {X 0,Y 459.564,Z 627.907,A -85,B 0,C 180,E1 -8005.616,E2 -8005.616} C_VEL
LIN {X 0,Y 459.583,Z 629.786,A -85,B 0,C 180,E1 -8006.494,E2 -8006.494} C_VEL
LIN {X 0,Y 459.584,Z 631.194,A -85,B 0,C 180,E1 -8007.372,E2 -8007.372} C_VEL
LIN {X 0,Y 459.521,Z 632.802,A -85,B 0,C 180,E1 -8009.125,E2 -8009.125} C_VEL
LIN {X 0,Y 459.53,Z 633.018,A -85,B 0,C 180,E1 -8010.001,E2 -8010.001} C_VEL
LIN {X 0,Y 459.521,Z 632.796,A -85,B 0,C 180,E1 -8010.877,E2 -8010.877} C_VEL
LIN {X 0,Y 459.584,Z 631.172,A -85,B 0,C 180,E1 -8012.631,E2 -8012.631} C_VEL
LIN {X 0,Y 459.584,Z 629.76,A -85,B 0,C 180,E1 -8013.508,E2 -8013.508} C_VEL
LIN {X 0,Y 459.618,Z 626.794,A -85,B 0,C 180,E1 -8014.825,E2 -8014.825} C_VEL
LIN {X 0,Y 459.715,Z 621.737,A -85,B 0,C 180,E1 -8016.432,E2 -8016.432} C_VEL
LIN {X 0,Y 459.908,Z 615.591,A -85,B 0,C 180,E1 -8017.906,E2 -8017.906} C_VEL
LIN {X 0,Y 460.223,Z 608.631,A -85,B 0,C 180,E1 -8019.228,E2 -8019.228} C_VEL
LIN {X 0,Y 460.597,Z 599.912,A -85,B 0,C 180,E1 -8020.552,E2 -8020.552} C_VEL
LIN {X 0,Y 461.128,Z 590.984,A -85,B 0,C 180,E1 -8021.652,E2 -8021.652} C_VEL
LIN {X 0,Y 461.564,Z 581.339,A -85,B 0,C 180,E1 -8022.629,E2 -8022.629} C_VEL
LIN {X 0,Y 462.084,Z 570.434,A -85,B 0,C 180,E1 -8023.525,E2 -8023.525} C_VEL
LIN {X 0,Y 462.618,Z 558.387,A -85,B 0,C 180,E1 -8024.293,E2 -8024.293} C_VEL
LIN {X 0,Y 463.117,Z 545.854,A -85,B 0,C 180,E1 -8024.895,E2 -8024.895} C_VEL
LIN {X 0,Y 463.504,Z 533.805,A -85,B 0,C 180,E1 -8025.304,E2 -8025.304} C_VEL
LIN {X 0,Y 463.817,Z 518.808,A -85,B 0,C 180,E1 -8025.603,E2 -8025.603} C_VEL
LIN {X 0,Y 464.444,Z 439.742,A -85,B 0,C 180,E1 -8026.864,E2 -8026.864} C_VEL
LIN {X 0,Y 461.376,Z 420.192,A -85,B 0,C 180,E1 -8027.326,E2 -8027.326} C_VEL
LIN {X 0,Y 462.126,Z 404.107,A -85,B 0,C 180,E1 -8030.243,E2 -8030.243} C_VEL
LIN {X 0,Y 462.962,Z 387.805,A -85,B 0,C 180,E1 -8033.248,E2 -8033.248} C_VEL
LIN {X 0,Y 462.083,Z 381.522,A -85,B 0,C 180,E1 -8034.486,E2 -8034.486} C_VEL
LIN {X 0,Y 460.563,Z 374.117,A -85,B 0,C 180,E1 -8036.025,E2 -8036.025} C_VEL
LIN {X 0,Y 460.561,Z 374.118,A -85,B 0,C 180,E1 -8038.233,E2 -8038.233} C_VEL
LIN {X 0,Y 460.527,Z 374.125,A -85,B 0,C 180,E1 -8041.284,E2 -8041.284} C_VEL
LIN {X 0,Y 460.538,Z 374.116,A -85,B 0,C 180,E1 -8044.506,E2 -8044.506} C_VEL
LIN {X 0,Y 460.507,Z 374.124,A -85,B 0,C 180,E1 -8047.624,E2 -8047.624} C_VEL
LIN {X 0,Y 460.547,Z 374.117,A -85,B 0,C 180,E1 -8050.27,E2 -8050.27} C_VEL
LIN {X 0,Y 460.506,Z 374.125,A -85,B 0,C 180,E1 -8053.376,E2 -8053.376} C_VEL
LIN {X 0,Y 460.506,Z 374.124,A -85,B 0,C 180,E1 -8056.625,E2 -8056.625} C_VEL
LIN {X 0,Y 460.544,Z 374.112,A -85,B 0,C 180,E1 -8059.731,E2 -8059.731} C_VEL
LIN {X 0,Y 460.505,Z 374.123,A -85,B 0,C 180,E1 -8062.524,E2 -8062.524} C_VEL
LIN {X 0,Y 460.551,Z 374.111,A -85,B 0,C 180,E1 -8065.624,E2 -8065.624} C_VEL
LIN {X 0,Y 460.543,Z 374.117,A -85,B 0,C 180,E1 -8068.745,E2 -8068.745} C_VEL
LIN {X 0,Y 460.587,Z 374.112,A -85,B 0,C 180,E1 -8072.254,E2 -8072.254} C_VEL
LIN {X 0,Y 460.545,Z 374.121,A -85,B 0,C 180,E1 -8074.705,E2 -8074.705} C_VEL
LIN {X 0,Y 460.516,Z 374.114,A -85,B 0,C 180,E1 -8077.572,E2 -8077.572} C_VEL
LIN {X 0,Y 460.574,Z 374.115,A -85,B 0,C 180,E1 -8080.385,E2 -8080.385} C_VEL
LIN {X 0,Y 460.57,Z 374.112,A -85,B 0,C 180,E1 -8083.146,E2 -8083.146} C_VEL
LIN {X 0,Y 460.56,Z 374.109,A -85,B 0,C 180,E1 -8085.868,E2 -8085.868} C_VEL
LIN {X 0,Y 460.616,Z 374.106,A -85,B 0,C 180,E1 -8088.559,E2 -8088.559} C_VEL
LIN {X 0,Y 460.701,Z 374.101,A -85,B 0,C 180,E1 -8092.109,E2 -8092.109} C_VEL
LIN {X 0,Y 460.703,Z 374.096,A -85,B 0,C 180,E1 -8094.748,E2 -8094.748} C_VEL
LIN {X 0,Y 460.806,Z 374.078,A -85,B 0,C 180,E1 -8097.378,E2 -8097.378} C_VEL
LIN {X 0,Y 460.858,Z 374.079,A -85,B 0,C 180,E1 -8100,E2 -8100} C_VEL
LIN {X 0,Y 460.806,Z 374.082,A -85,B 0,C 180,E1 -8102.623,E2 -8102.623} C_VEL
LIN {X 0,Y 460.716,Z 374.096,A -85,B 0,C 180,E1 -8106.13,E2 -8106.13} C_VEL
LIN {X 0,Y 460.634,Z 374.103,A -85,B 0,C 180,E1 -8108.776,E2 -8108.776} C_VEL
LIN {X 0,Y 460.62,Z 374.107,A -85,B 0,C 180,E1 -8112.445,E2 -8112.445} C_VEL
LIN {X 0,Y 460.606,Z 374.112,A -85,B 0,C 180,E1 -8115.997,E2 -8115.997} C_VEL
LIN {X 0,Y 460.577,Z 374.112,A -85,B 0,C 180,E1 -8118.902,E2 -8118.902} C_VEL
LIN {X 0,Y 460.522,Z 374.124,A -85,B 0,C 180,E1 -8121.485,E2 -8121.485} C_VEL
LIN {X 0,Y 460.537,Z 374.118,A -85,B 0,C 180,E1 -8124.333,E2 -8124.333} C_VEL
LIN {X 0,Y 460.578,Z 374.115,A -85,B 0,C 180,E1 -8127.244,E2 -8127.244} C_VEL
LIN {X 0,Y 460.631,Z 374.303,A -85,B 0,C 180,E1 -8129.713,E2 -8129.713} C_VEL
LIN {X 0,Y 462.177,Z 383.225,A -85,B 0,C 180,E1 -8131.795,E2 -8131.795} C_VEL
LIN {X 0,Y 461.633,Z 397.087,A -85,B 0,C 180,E1 -8134.772,E2 -8134.772} C_VEL
LIN {X 0,Y 464.652,Z 412.877,A -85,B 0,C 180,E1 -8135.154,E2 -8135.154} C_VEL
LIN {X 0,Y 463.708,Z 504.058,A -85,B 0,C 180,E1 -8136.627,E2 -8136.627} C_VEL
LIN {X 0,Y 463.39,Z 517.521,A -85,B 0,C 180,E1 -8137.028,E2 -8137.028} C_VEL
LIN {X 0,Y 463.048,Z 529.929,A -85,B 0,C 180,E1 -8137.577,E2 -8137.577} C_VEL
LIN {X 0,Y 462.589,Z 541.286,A -85,B 0,C 180,E1 -8138.253,E2 -8138.253} C_VEL
LIN {X 0,Y 462.051,Z 552.732,A -85,B 0,C 180,E1 -8139.127,E2 -8139.127} C_VEL
LIN {X 0,Y 461.486,Z 563.559,A -85,B 0,C 180,E1 -8140.166,E2 -8140.166} C_VEL
LIN {X 0,Y 460.98,Z 572.946,A -85,B 0,C 180,E1 -8141.291,E2 -8141.291} C_VEL
LIN {X 0,Y 460.589,Z 581.343,A -85,B 0,C 180,E1 -8142.532,E2 -8142.532} C_VEL
LIN {X 0,Y 460.189,Z 588.129,A -85,B 0,C 180,E1 -8143.76,E2 -8143.76} C_VEL
LIN {X 0,Y 459.914,Z 593.643,A -85,B 0,C 180,E1 -8144.988,E2 -8144.988} C_VEL
LIN {X 0,Y 459.729,Z 599.076,A -85,B 0,C 180,E1 -8146.533,E2 -8146.533} C_VEL
LIN {X 0,Y 459.626,Z 602.192,A -85,B 0,C 180,E1 -8147.716,E2 -8147.716} C_VEL
LIN {X 0,Y 459.509,Z 604.468,A -85,B 0,C 180,E1 -8148.877,E2 -8148.877} C_VEL
LIN {X 0,Y 459.455,Z 606.024,A -85,B 0,C 180,E1 -8150.024,E2 -8150.024} C_VEL
LIN {X 0,Y 459.408,Z 606.92,A -85,B 0,C 180,E1 -8151.279,E2 -8151.279} C_VEL
LIN {X 0,Y 459.409,Z 606.946,A -85,B 0,C 180,E1 -8152.702,E2 -8152.702} C_VEL
LIN {X 0,Y 459.466,Z 605.503,A -85,B 0,C 180,E1 -8154.461,E2 -8154.461} C_VEL
LIN {X 0,Y 459.622,Z 602.629,A -85,B 0,C 180,E1 -8156.139,E2 -8156.139} C_VEL
LIN {X 0,Y 459.77,Z 598.645,A -85,B 0,C 180,E1 -8157.655,E2 -8157.655} C_VEL
LIN {X 0,Y 459.92,Z 594.656,A -85,B 0,C 180,E1 -8158.807,E2 -8158.807} C_VEL
LIN {X 0,Y 459.37,Z 592.109,A -85,B 0,C 180,E1 -8159.469,E2 -8159.469} C_VEL
LIN {X 0,Y 456.76,Z 587.533,A -85,B 0,C 180,E1 -8160.521,E2 -8160.521} C_VEL
LIN {X 0,Y 454.179,Z 582.27,A -85,B 0,C 180,E1 -8161.531,E2 -8161.531} C_VEL
LIN {X 0,Y 453.677,Z 578.645,A -85,B 0,C 180,E1 -8162.119,E2 -8162.119} C_VEL
LIN {X 0,Y 454.106,Z 569.914,A -85,B 0,C 180,E1 -8163.331,E2 -8163.331} C_VEL
LIN {X 0,Y 454.694,Z 559.72,A -85,B 0,C 180,E1 -8164.477,E2 -8164.477} C_VEL
LIN {X 0,Y 455.257,Z 548.933,A -85,B 0,C 180,E1 -8165.445,E2 -8165.445} C_VEL
LIN {X 0,Y 455.769,Z 537.597,A -85,B 0,C 180,E1 -8166.252,E2 -8166.252} C_VEL
LIN {X 0,Y 456.207,Z 525.286,A -85,B 0,C 180,E1 -8166.928,E2 -8166.928} C_VEL
LIN {X 0,Y 456.607,Z 512.874,A -85,B 0,C 180,E1 -8167.414,E2 -8167.414} C_VEL
LIN {X 0,Y 456.846,Z 500.133,A -85,B 0,C 180,E1 -8167.738,E2 -8167.738} C_VEL
LIN {X 0,Y 457.582,Z 412.374,A -85,B 0,C 180,E1 -8169.165,E2 -8169.165} C_VEL
LIN {X 0,Y 454.56,Z 396.623,A -85,B 0,C 180,E1 -8169.553,E2 -8169.553} C_VEL
LIN {X 0,Y 455.107,Z 384.281,A -85,B 0,C 180,E1 -8172.241,E2 -8172.241} C_VEL
LIN {X 0,Y 453.591,Z 374.987,A -85,B 0,C 180,E1 -8174.404,E2 -8174.404} C_VEL
LIN {X 0,Y 453.569,Z 374.984,A -85,B 0,C 180,E1 -8177.47,E2 -8177.47} C_VEL
LIN {X 0,Y 453.597,Z 374.98,A -85,B 0,C 180,E1 -8181.086,E2 -8181.086} C_VEL
LIN {X 0,Y 453.656,Z 374.972,A -85,B 0,C 180,E1 -8183.773,E2 -8183.773} C_VEL
LIN {X 0,Y 453.749,Z 374.96,A -85,B 0,C 180,E1 -8187.336,E2 -8187.336} C_VEL
LIN {X 0,Y 453.827,Z 374.953,A -85,B 0,C 180,E1 -8189.999,E2 -8189.999} C_VEL
LIN {X 0,Y 453.768,Z 374.96,A -85,B 0,C 180,E1 -8192.662,E2 -8192.662} C_VEL
LIN {X 0,Y 453.68,Z 374.976,A -85,B 0,C 180,E1 -8196.224,E2 -8196.224} C_VEL
LIN {X 0,Y 453.593,Z 374.979,A -85,B 0,C 180,E1 -8198.912,E2 -8198.912} C_VEL
LIN {X 0,Y 453.565,Z 374.985,A -85,B 0,C 180,E1 -8202.527,E2 -8202.527} C_VEL
LIN {X 0,Y 453.557,Z 374.989,A -85,B 0,C 180,E1 -8206.194,E2 -8206.194} C_VEL
LIN {X 0,Y 453.521,Z 374.988,A -85,B 0,C 180,E1 -8209.039,E2 -8209.039} C_VEL
LIN {X 0,Y 453.476,Z 375.001,A -85,B 0,C 180,E1 -8211.835,E2 -8211.835} C_VEL
LIN {X 0,Y 453.499,Z 374.991,A -85,B 0,C 180,E1 -8214.734,E2 -8214.734} C_VEL
LIN {X 0,Y 453.537,Z 374.992,A -85,B 0,C 180,E1 -8217.96,E2 -8217.96} C_VEL
LIN {X 0,Y 453.481,Z 374.993,A -85,B 0,C 180,E1 -8220.758,E2 -8220.758} C_VEL
LIN {X 0,Y 453.475,Z 374.999,A -85,B 0,C 180,E1 -8223.911,E2 -8223.911} C_VEL
LIN {X 0,Y 453.468,Z 374.997,A -85,B 0,C 180,E1 -8227.186,E2 -8227.186} C_VEL
LIN {X 0,Y 453.527,Z 374.993,A -85,B 0,C 180,E1 -8229.444,E2 -8229.444} C_VEL
LIN {X 0,Y 453.462,Z 374.997,A -85,B 0,C 180,E1 -8232.993,E2 -8232.993} C_VEL
LIN {X 0,Y 453.508,Z 374.995,A -85,B 0,C 180,E1 -8236.363,E2 -8236.363} C_VEL
LIN {X 0,Y 453.542,Z 375.178,A -85,B 0,C 180,E1 -8236.479,E2 -8236.479} C_VEL
LIN {X 0,Y 454.706,Z 382.058,A -85,B 0,C 180,E1 -8237.891,E2 -8237.891} C_VEL
LIN {X 0,Y 454.455,Z 396.032,A -85,B 0,C 180,E1 -8240.6,E2 -8240.6} C_VEL
LIN {X 0,Y 457.532,Z 413.126,A -85,B 0,C 180,E1 -8241.016,E2 -8241.016} C_VEL
LIN {X 0,Y 456.482,Z 504.19,A -85,B 0,C 180,E1 -8242.579,E2 -8242.579} C_VEL
LIN {X 0,Y 456.204,Z 516.072,A -85,B 0,C 180,E1 -8242.934,E2 -8242.934} C_VEL
LIN {X 0,Y 455.86,Z 528.311,A -85,B 0,C 180,E1 -8243.467,E2 -8243.467} C_VEL
LIN {X 0,Y 455.342,Z 540.961,A -85,B 0,C 180,E1 -8244.215,E2 -8244.215} C_VEL
LIN {X 0,Y 454.904,Z 550.889,A -85,B 0,C 180,E1 -8244.964,E2 -8244.964} C_VEL
LIN {X 0,Y 454.402,Z 560.966,A -85,B 0,C 180,E1 -8245.898,E2 -8245.898} C_VEL
LIN {X 0,Y 453.96,Z 570.097,A -85,B 0,C 180,E1 -8246.94,E2 -8246.94} C_VEL
LIN {X 0,Y 453.518,Z 579.156,A -85,B 0,C 180,E1 -8248.204,E2 -8248.204} C_VEL
LIN {X 0,Y 453.142,Z 586.539,A -85,B 0,C 180,E1 -8249.473,E2 -8249.473} C_VEL
LIN {X 0,Y 452.881,Z 592.67,A -85,B 0,C 180,E1 -8250.784,E2 -8250.784} C_VEL
LIN {X 0,Y 452.682,Z 598.019,A -85,B 0,C 180,E1 -8252.241,E2 -8252.241} C_VEL
LIN {X 0,Y 452.516,Z 602.116,A -85,B 0,C 180,E1 -8253.728,E2 -8253.728} C_VEL
LIN {X 0,Y 452.365,Z 604.934,A -85,B 0,C 180,E1 -8255.198,E2 -8255.198} C_VEL
LIN {X 0,Y 452.319,Z 606.393,A -85,B 0,C 180,E1 -8256.448,E2 -8256.448} C_VEL
LIN {X 0,Y 452.293,Z 607.121,A -85,B 0,C 180,E1 -8258.104,E2 -8258.104} C_VEL
LIN {X 0,Y 452.362,Z 606.858,A -85,B 0,C 180,E1 -8259.063,E2 -8259.063} C_VEL
LIN {X 0,Y 452.366,Z 606.165,A -85,B 0,C 180,E1 -8260.014,E2 -8260.014} C_VEL
LIN {X 0,Y 452.449,Z 604.372,A -85,B 0,C 180,E1 -8261.352,E2 -8261.352} C_VEL
LIN {X 0,Y 452.583,Z 601.257,A -85,B 0,C 180,E1 -8262.84,E2 -8262.84} C_VEL
LIN {X 0,Y 452.702,Z 597.064,A -85,B 0,C 180,E1 -8264.258,E2 -8264.258} C_VEL
LIN {X 0,Y 453.038,Z 590.734,A -85,B 0,C 180,E1 -8265.858,E2 -8265.858} C_VEL
LIN {X 0,Y 453.33,Z 583.756,A -85,B 0,C 180,E1 -8267.237,E2 -8267.237} C_VEL
LIN {X 0,Y 453.809,Z 574.959,A -85,B 0,C 180,E1 -8268.612,E2 -8268.612} C_VEL
LIN {X 0,Y 454.26,Z 565.971,A -85,B 0,C 180,E1 -8269.751,E2 -8269.751} C_VEL
LIN {X 0,Y 454.802,Z 556.028,A -85,B 0,C 180,E1 -8270.774,E2 -8270.774} C_VEL
LIN {X 0,Y 455.433,Z 543.992,A -85,B 0,C 180,E1 -8271.76,E2 -8271.76} C_VEL
LIN {X 0,Y 455.925,Z 532.933,A -85,B 0,C 180,E1 -8272.471,E2 -8272.471} C_VEL
LIN {X 0,Y 456.271,Z 520.21,A -85,B 0,C 180,E1 -8273.088,E2 -8273.088} C_VEL
LIN {X 0,Y 456.63,Z 507.785,A -85,B 0,C 180,E1 -8273.51,E2 -8273.51} C_VEL
LIN {X 0,Y 456.782,Z 492.868,A -85,B 0,C 180,E1 -8273.817,E2 -8273.817} C_VEL
LIN {X 0,Y 457.811,Z 412.593,A -85,B 0,C 180,E1 -8275.212,E2 -8275.212} C_VEL
LIN {X 0,Y 454.615,Z 396.236,A -85,B 0,C 180,E1 -8275.678,E2 -8275.678} C_VEL
LIN {X 0,Y 454.872,Z 383.032,A -85,B 0,C 180,E1 -8278.229,E2 -8278.229} C_VEL
LIN {X 0,Y 453.805,Z 374.96,A -85,B 0,C 180,E1 -8279.834,E2 -8279.834} C_VEL
LIN {X 0,Y 453.756,Z 374.967,A -85,B 0,C 180,E1 -8282.663,E2 -8282.663} C_VEL
LIN {X 0,Y 453.667,Z 374.978,A -85,B 0,C 180,E1 -8286.225,E2 -8286.225} C_VEL
LIN {X 0,Y 453.583,Z 374.985,A -85,B 0,C 180,E1 -8288.914,E2 -8288.914} C_VEL
LIN {X 0,Y 453.59,Z 374.985,A -85,B 0,C 180,E1 -8292.551,E2 -8292.551} C_VEL
LIN {X 0,Y 453.545,Z 374.993,A -85,B 0,C 180,E1 -8296.196,E2 -8296.196} C_VEL
LIN {X 0,Y 453.51,Z 374.992,A -85,B 0,C 180,E1 -8299.042,E2 -8299.042} C_VEL
LIN {X 0,Y 453.495,Z 374.998,A -85,B 0,C 180,E1 -8301.835,E2 -8301.835} C_VEL
LIN {X 0,Y 453.521,Z 374.99,A -85,B 0,C 180,E1 -8304.734,E2 -8304.734} C_VEL
LIN {X 0,Y 453.529,Z 374.993,A -85,B 0,C 180,E1 -8307.962,E2 -8307.962} C_VEL
LIN {X 0,Y 453.474,Z 374.996,A -85,B 0,C 180,E1 -8310.76,E2 -8310.76} C_VEL
LIN {X 0,Y 453.469,Z 375,A -85,B 0,C 180,E1 -8313.913,E2 -8313.913} C_VEL
LIN {X 0,Y 453.462,Z 375.001,A -85,B 0,C 180,E1 -8317.189,E2 -8317.189} C_VEL
LIN {X 0,Y 453.509,Z 374.997,A -85,B 0,C 180,E1 -8319.448,E2 -8319.448} C_VEL
LIN {X 0,Y 453.461,Z 375,A -85,B 0,C 180,E1 -8322.995,E2 -8322.995} C_VEL
LIN {X 0,Y 453.467,Z 374.997,A -85,B 0,C 180,E1 -8325.781,E2 -8325.781} C_VEL
LIN {X 0,Y 453.475,Z 374.995,A -85,B 0,C 180,E1 -8328.211,E2 -8328.211} C_VEL
LIN {X 0,Y 453.505,Z 374.996,A -85,B 0,C 180,E1 -8330.792,E2 -8330.792} C_VEL
LIN {X 0,Y 453.452,Z 374.998,A -85,B 0,C 180,E1 -8333.919,E2 -8333.919} C_VEL
LIN {X 0,Y 453.479,Z 374.999,A -85,B 0,C 180,E1 -8337.153,E2 -8337.153} C_VEL
LIN {X 0,Y 453.511,Z 374.994,A -85,B 0,C 180,E1 -8340.273,E2 -8340.273} C_VEL
LIN {X 0,Y 453.535,Z 374.993,A -85,B 0,C 180,E1 -8343.297,E2 -8343.297} C_VEL
LIN {X 0,Y 453.577,Z 375.107,A -85,B 0,C 180,E1 -8343.837,E2 -8343.837} C_VEL
LIN {X 0,Y 455.937,Z 387.613,A -85,B 0,C 180,E1 -8346.375,E2 -8346.375} C_VEL
LIN {X 0,Y 455.382,Z 400.225,A -85,B 0,C 180,E1 -8348.737,E2 -8348.737} C_VEL
LIN {X 0,Y 454.606,Z 416.601,A -85,B 0,C 180,E1 -8351.758,E2 -8351.758} C_VEL
LIN {X 0,Y 454.421,Z 420.492,A -85,B 0,C 180,E1 -8352.47,E2 -8352.47} C_VEL
LIN {X 0,Y 457.611,Z 441.414,A -85,B 0,C 180,E1 -8352.945,E2 -8352.945} C_VEL
LIN {X 0,Y 456.734,Z 529.107,A -85,B 0,C 180,E1 -8354.38,E2 -8354.38} C_VEL
LIN {X 0,Y 456.326,Z 542.909,A -85,B 0,C 180,E1 -8354.795,E2 -8354.795} C_VEL
LIN {X 0,Y 455.869,Z 554.78,A -85,B 0,C 180,E1 -8355.322,E2 -8355.322} C_VEL
LIN {X 0,Y 455.321,Z 566.824,A -85,B 0,C 180,E1 -8356.045,E2 -8356.045} C_VEL
LIN {X 0,Y 454.752,Z 578.184,A -85,B 0,C 180,E1 -8356.925,E2 -8356.925} C_VEL
LIN {X 0,Y 454.259,Z 588.722,A -85,B 0,C 180,E1 -8357.946,E2 -8357.946} C_VEL
LIN {X 0,Y 453.706,Z 598.039,A -85,B 0,C 180,E1 -8359.063,E2 -8359.063} C_VEL
LIN {X 0,Y 453.235,Z 607.08,A -85,B 0,C 180,E1 -8360.406,E2 -8360.406} C_VEL
LIN {X 0,Y 452.909,Z 614.361,A -85,B 0,C 180,E1 -8361.749,E2 -8361.749} C_VEL
LIN {X 0,Y 452.718,Z 619.275,A -85,B 0,C 180,E1 -8362.867,E2 -8362.867} C_VEL
LIN {X 0,Y 452.564,Z 624.047,A -85,B 0,C 180,E1 -8364.208,E2 -8364.208} C_VEL
LIN {X 0,Y 452.486,Z 627.693,A -85,B 0,C 180,E1 -8365.547,E2 -8365.547} C_VEL
LIN {X 0,Y 452.48,Z 629.575,A -85,B 0,C 180,E1 -8366.439,E2 -8366.439} C_VEL
LIN {X 0,Y 452.507,Z 630.988,A -85,B 0,C 180,E1 -8367.331,E2 -8367.331} C_VEL
LIN {X 0,Y 452.428,Z 632.599,A -85,B 0,C 180,E1 -8369.111,E2 -8369.111} C_VEL
LIN {X 0,Y 452.434,Z 632.817,A -85,B 0,C 180,E1 -8370.001,E2 -8370.001} C_VEL
LIN {X 0,Y 452.428,Z 632.597,A -85,B 0,C 180,E1 -8370.891,E2 -8370.891} C_VEL
LIN {X 0,Y 452.508,Z 630.975,A -85,B 0,C 180,E1 -8372.672,E2 -8372.672} C_VEL
LIN {X 0,Y 452.48,Z 629.563,A -85,B 0,C 180,E1 -8373.563,E2 -8373.563} C_VEL
LIN {X 0,Y 452.547,Z 626.598,A -85,B 0,C 180,E1 -8374.901,E2 -8374.901} C_VEL
LIN {X 0,Y 452.611,Z 622.042,A -85,B 0,C 180,E1 -8376.397,E2 -8376.397} C_VEL
LIN {X 0,Y 452.816,Z 616.419,A -85,B 0,C 180,E1 -8377.806,E2 -8377.806} C_VEL
LIN {X 0,Y 453.11,Z 609.685,A -85,B 0,C 180,E1 -8379.149,E2 -8379.149} C_VEL
LIN {X 0,Y 453.499,Z 601.332,A -85,B 0,C 180,E1 -8380.493,E2 -8380.493} C_VEL
LIN {X 0,Y 454.029,Z 592.759,A -85,B 0,C 180,E1 -8381.61,E2 -8381.61} C_VEL
LIN {X 0,Y 454.552,Z 583.047,A -85,B 0,C 180,E1 -8382.645,E2 -8382.645} C_VEL
LIN {X 0,Y 455.078,Z 571.696,A -85,B 0,C 180,E1 -8383.623,E2 -8383.623} C_VEL
LIN {X 0,Y 455.644,Z 560.189,A -85,B 0,C 180,E1 -8384.403,E2 -8384.403} C_VEL
LIN {X 0,Y 456.227,Z 546.99,A -85,B 0,C 180,E1 -8385.068,E2 -8385.068} C_VEL
LIN {X 0,Y 456.647,Z 534.585,A -85,B 0,C 180,E1 -8385.511,E2 -8385.511} C_VEL
LIN {X 0,Y 456.972,Z 522.263,A -85,B 0,C 180,E1 -8385.786,E2 -8385.786} C_VEL
LIN {X 0,Y 457.564,Z 439.845,A -85,B 0,C 180,E1 -8387.128,E2 -8387.128} C_VEL
LIN {X 0,Y 454.42,Z 420.029,A -85,B 0,C 180,E1 -8387.6,E2 -8387.6} C_VEL
LIN {X 0,Y 455.158,Z 403.971,A -85,B 0,C 180,E1 -8390.567,E2 -8390.567} C_VEL
LIN {X 0,Y 456.042,Z 388.943,A -85,B 0,C 180,E1 -8393.381,E2 -8393.381} C_VEL
LIN {X 0,Y 455.107,Z 382.689,A -85,B 0,C 180,E1 -8394.643,E2 -8394.643} C_VEL
LIN {X 0,Y 453.549,Z 374.99,A -85,B 0,C 180,E1 -8396.261,E2 -8396.261} C_VEL
LIN {X 0,Y 453.517,Z 374.996,A -85,B 0,C 180,E1 -8398.712,E2 -8398.712} C_VEL
LIN {X 0,Y 453.47,Z 375,A -85,B 0,C 180,E1 -8401.8,E2 -8401.8} C_VEL
LIN {X 0,Y 453.486,Z 374.999,A -85,B 0,C 180,E1 -8404.99,E2 -8404.99} C_VEL
LIN {X 0,Y 453.47,Z 374.999,A -85,B 0,C 180,E1 -8408.312,E2 -8408.312} C_VEL
LIN {X 0,Y 453.499,Z 374.997,A -85,B 0,C 180,E1 -8410.609,E2 -8410.609} C_VEL
LIN {X 0,Y 453.462,Z 375.004,A -85,B 0,C 180,E1 -8413.245,E2 -8413.245} C_VEL
LIN {X 0,Y 453.472,Z 374.997,A -85,B 0,C 180,E1 -8415.78,E2 -8415.78} C_VEL
LIN {X 0,Y 453.484,Z 374.994,A -85,B 0,C 180,E1 -8418.21,E2 -8418.21} C_VEL
LIN {X 0,Y 453.497,Z 374.996,A -85,B 0,C 180,E1 -8420.794,E2 -8420.794} C_VEL
LIN {X 0,Y 453.459,Z 374.996,A -85,B 0,C 180,E1 -8423.918,E2 -8423.918} C_VEL
LIN {X 0,Y 453.488,Z 374.996,A -85,B 0,C 180,E1 -8427.152,E2 -8427.152} C_VEL
LIN {X 0,Y 453.48,Z 374.992,A -85,B 0,C 180,E1 -8430.269,E2 -8430.269} C_VEL
LIN {X 0,Y 453.507,Z 374.988,A -85,B 0,C 180,E1 -8433.294,E2 -8433.294} C_VEL
LIN {X 0,Y 453.503,Z 374.995,A -85,B 0,C 180,E1 -8436.239,E2 -8436.239} C_VEL
LIN {X 0,Y 453.488,Z 374.995,A -85,B 0,C 180,E1 -8439.118,E2 -8439.118} C_VEL
LIN {X 0,Y 453.516,Z 374.987,A -85,B 0,C 180,E1 -8441.945,E2 -8441.945} C_VEL
LIN {X 0,Y 453.545,Z 374.984,A -85,B 0,C 180,E1 -8444.727,E2 -8444.727} C_VEL
LIN {X 0,Y 453.565,Z 374.986,A -85,B 0,C 180,E1 -8448.379,E2 -8448.379} C_VEL
LIN {X 0,Y 453.658,Z 374.977,A -85,B 0,C 180,E1 -8451.985,E2 -8451.985} C_VEL
LIN {X 0,Y 453.677,Z 374.972,A -85,B 0,C 180,E1 -8454.667,E2 -8454.667} C_VEL
LIN {X 0,Y 453.75,Z 374.956,A -85,B 0,C 180,E1 -8457.337,E2 -8457.337} C_VEL
LIN {X 0,Y 453.829,Z 374.955,A -85,B 0,C 180,E1 -8460,E2 -8460} C_VEL
LIN {X 0,Y 453.75,Z 374.961,A -85,B 0,C 180,E1 -8462.663,E2 -8462.663} C_VEL
LIN {X 0,Y 453.683,Z 374.971,A -85,B 0,C 180,E1 -8466.225,E2 -8466.225} C_VEL
LIN {X 0,Y 453.598,Z 374.98,A -85,B 0,C 180,E1 -8468.913,E2 -8468.913} C_VEL
LIN {X 0,Y 453.57,Z 374.984,A -85,B 0,C 180,E1 -8472.529,E2 -8472.529} C_VEL
LIN {X 0,Y 453.551,Z 374.989,A -85,B 0,C 180,E1 -8476.196,E2 -8476.196} C_VEL
LIN {X 0,Y 453.526,Z 374.992,A -85,B 0,C 180,E1 -8479.04,E2 -8479.04} C_VEL
LIN {X 0,Y 453.483,Z 374.999,A -85,B 0,C 180,E1 -8481.836,E2 -8481.836} C_VEL
LIN {X 0,Y 453.507,Z 374.994,A -85,B 0,C 180,E1 -8484.735,E2 -8484.735} C_VEL
LIN {X 0,Y 453.54,Z 374.991,A -85,B 0,C 180,E1 -8487.96,E2 -8487.96} C_VEL
LIN {X 0,Y 453.546,Z 375.126,A -85,B 0,C 180,E1 -8489.472,E2 -8489.472} C_VEL
LIN {X 0,Y 455.212,Z 384.346,A -85,B 0,C 180,E1 -8491.663,E2 -8491.663} C_VEL
LIN {X 0,Y 454.686,Z 397.094,A -85,B 0,C 180,E1 -8494.479,E2 -8494.479} C_VEL
LIN {X 0,Y 457.885,Z 414.178,A -85,B 0,C 180,E1 -8494.906,E2 -8494.906} C_VEL
LIN {X 0,Y 456.885,Z 504.725,A -85,B 0,C 180,E1 -8496.401,E2 -8496.401} C_VEL
LIN {X 0,Y 456.556,Z 517.878,A -85,B 0,C 180,E1 -8496.802,E2 -8496.802} C_VEL
LIN {X 0,Y 456.186,Z 529.998,A -85,B 0,C 180,E1 -8497.345,E2 -8497.345} C_VEL
LIN {X 0,Y 455.711,Z 541.5,A -85,B 0,C 180,E1 -8498.039,E2 -8498.039} C_VEL
LIN {X 0,Y 455.137,Z 552.106,A -85,B 0,C 180,E1 -8498.852,E2 -8498.852} C_VEL
LIN {X 0,Y 454.567,Z 563.259,A -85,B 0,C 180,E1 -8499.926,E2 -8499.926} C_VEL
LIN {X 0,Y 454.006,Z 572.585,A -85,B 0,C 180,E1 -8501.042,E2 -8501.042} C_VEL
LIN {X 0,Y 453.616,Z 580.252,A -85,B 0,C 180,E1 -8502.164,E2 -8502.164} C_VEL
LIN {X 0,Y 453.18,Z 587.693,A -85,B 0,C 180,E1 -8503.497,E2 -8503.497} C_VEL
LIN {X 0,Y 452.839,Z 594.519,A -85,B 0,C 180,E1 -8505.04,E2 -8505.04} C_VEL
LIN {X 0,Y 452.671,Z 598.839,A -85,B 0,C 180,E1 -8506.299,E2 -8506.299} C_VEL
LIN {X 0,Y 452.569,Z 602.065,A -85,B 0,C 180,E1 -8507.505,E2 -8507.505} C_VEL
LIN {X 0,Y 452.373,Z 605.363,A -85,B 0,C 180,E1 -8509.268,E2 -8509.268} C_VEL
LIN {X 0,Y 452.312,Z 606.973,A -85,B 0,C 180,E1 -8510.978,E2 -8510.978} C_VEL
LIN {X 0,Y 452.318,Z 607.148,A -85,B 0,C 180,E1 -8512.7,E2 -8512.7} C_VEL
LIN {X 0,Y 452.351,Z 606.359,A -85,B 0,C 180,E1 -8513.892,E2 -8513.892} C_VEL
LIN {X 0,Y 452.442,Z 604.335,A -85,B 0,C 180,E1 -8515.414,E2 -8515.414} C_VEL
LIN {X 0,Y 452.612,Z 600.703,A -85,B 0,C 180,E1 -8517.079,E2 -8517.079} C_VEL
LIN {X 0,Y 452.804,Z 595.907,A -85,B 0,C 180,E1 -8518.612,E2 -8518.612} C_VEL
LIN {X 0,Y 453.048,Z 590.341,A -85,B 0,C 180,E1 -8519.98,E2 -8519.98} C_VEL
LIN {X 0,Y 453.405,Z 583.73,A -85,B 0,C 180,E1 -8521.28,E2 -8521.28} C_VEL
LIN {X 0,Y 453.677,Z 578.645,A -85,B 0,C 180,E1 -8522.119,E2 -8522.119} C_VEL
LIN {X 0,Y 453.189,Z 574.896,A -85,B 0,C 180,E1 -8522.689,E2 -8522.689} C_VEL
LIN {X 0,Y 449.598,Z 565.869,A -85,B 0,C 180,E1 -8523.952,E2 -8523.952} C_VEL
LIN {X 0,Y 448.041,Z 560.182,A -85,B 0,C 180,E1 -8524.624,E2 -8524.624} C_VEL
LIN {X 0,Y 447.923,Z 557.075,A -85,B 0,C 180,E1 -8524.938,E2 -8524.938} C_VEL
LIN {X 0,Y 448.461,Z 546.267,A -85,B 0,C 180,E1 -8525.871,E2 -8525.871} C_VEL
LIN {X 0,Y 449.013,Z 534.637,A -85,B 0,C 180,E1 -8526.658,E2 -8526.658} C_VEL
LIN {X 0,Y 449.469,Z 522.042,A -85,B 0,C 180,E1 -8527.301,E2 -8527.301} C_VEL
LIN {X 0,Y 449.831,Z 509.52,A -85,B 0,C 180,E1 -8527.753,E2 -8527.753} C_VEL
LIN {X 0,Y 450.074,Z 495.916,A -85,B 0,C 180,E1 -8528.049,E2 -8528.049} C_VEL
LIN {X 0,Y 450.797,Z 413.294,A -85,B 0,C 180,E1 -8529.409,E2 -8529.409} C_VEL
LIN {X 0,Y 447.609,Z 396.757,A -85,B 0,C 180,E1 -8529.834,E2 -8529.834} C_VEL
LIN {X 0,Y 448.105,Z 385.035,A -85,B 0,C 180,E1 -8532.426,E2 -8532.426} C_VEL
LIN {X 0,Y 446.547,Z 375.864,A -85,B 0,C 180,E1 -8534.597,E2 -8534.597} C_VEL
LIN {X 0,Y 446.523,Z 375.864,A -85,B 0,C 180,E1 -8538.192,E2 -8538.192} C_VEL
LIN {X 0,Y 446.543,Z 375.86,A -85,B 0,C 180,E1 -8540.944,E2 -8540.944} C_VEL
LIN {X 0,Y 446.624,Z 375.847,A -85,B 0,C 180,E1 -8543.675,E2 -8543.675} C_VEL
LIN {X 0,Y 446.696,Z 375.838,A -85,B 0,C 180,E1 -8547.293,E2 -8547.293} C_VEL
LIN {X 0,Y 446.797,Z 375.829,A -85,B 0,C 180,E1 -8549.999,E2 -8549.999} C_VEL
LIN {X 0,Y 446.712,Z 375.839,A -85,B 0,C 180,E1 -8552.704,E2 -8552.704} C_VEL
LIN {X 0,Y 446.65,Z 375.85,A -85,B 0,C 180,E1 -8556.322,E2 -8556.322} C_VEL
LIN {X 0,Y 446.539,Z 375.858,A -85,B 0,C 180,E1 -8559.054,E2 -8559.054} C_VEL
LIN {X 0,Y 446.523,Z 375.861,A -85,B 0,C 180,E1 -8562.728,E2 -8562.728} C_VEL
LIN {X 0,Y 446.52,Z 375.865,A -85,B 0,C 180,E1 -8566.237,E2 -8566.237} C_VEL
LIN {X 0,Y 446.469,Z 375.867,A -85,B 0,C 180,E1 -8569.302,E2 -8569.302} C_VEL
LIN {X 0,Y 446.417,Z 375.877,A -85,B 0,C 180,E1 -8572.198,E2 -8572.198} C_VEL
LIN {X 0,Y 446.442,Z 375.871,A -85,B 0,C 180,E1 -8575.152,E2 -8575.152} C_VEL
LIN {X 0,Y 446.482,Z 375.868,A -85,B 0,C 180,E1 -8578.177,E2 -8578.177} C_VEL
LIN {X 0,Y 446.428,Z 375.874,A -85,B 0,C 180,E1 -8581.298,E2 -8581.298} C_VEL
LIN {X 0,Y 446.427,Z 375.872,A -85,B 0,C 180,E1 -8584.521,E2 -8584.521} C_VEL
LIN {X 0,Y 446.434,Z 375.873,A -85,B 0,C 180,E1 -8588.082,E2 -8588.082} C_VEL
LIN {X 0,Y 446.439,Z 375.871,A -85,B 0,C 180,E1 -8590.919,E2 -8590.919} C_VEL
LIN {X 0,Y 446.417,Z 375.879,A -85,B 0,C 180,E1 -8593.842,E2 -8593.842} C_VEL
LIN {X 0,Y 446.487,Z 375.933,A -85,B 0,C 180,E1 -8596.312,E2 -8596.312} C_VEL
LIN {X 0,Y 447.73,Z 383.478,A -85,B 0,C 180,E1 -8597.868,E2 -8597.868} C_VEL
LIN {X 0,Y 447.467,Z 395.942,A -85,B 0,C 180,E1 -8600.336,E2 -8600.336} C_VEL
LIN {X 0,Y 450.698,Z 413.765,A -85,B 0,C 180,E1 -8600.781,E2 -8600.781} C_VEL
LIN {X 0,Y 449.6,Z 504.292,A -85,B 0,C 180,E1 -8602.366,E2 -8602.366} C_VEL
LIN {X 0,Y 449.295,Z 517.094,A -85,B 0,C 180,E1 -8602.759,E2 -8602.759} C_VEL
LIN {X 0,Y 448.817,Z 530.624,A -85,B 0,C 180,E1 -8603.383,E2 -8603.383} C_VEL
LIN {X 0,Y 448.339,Z 542.69,A -85,B 0,C 180,E1 -8604.135,E2 -8604.135} C_VEL
LIN {X 0,Y 447.795,Z 554.03,A -85,B 0,C 180,E1 -8605.05,E2 -8605.05} C_VEL
LIN {X 0,Y 447.281,Z 564.286,A -85,B 0,C 180,E1 -8606.08,E2 -8606.08} C_VEL
LIN {X 0,Y 446.794,Z 572.892,A -85,B 0,C 180,E1 -8607.133,E2 -8607.133} C_VEL
LIN {X 0,Y 446.4,Z 581.642,A -85,B 0,C 180,E1 -8608.455,E2 -8608.455} C_VEL
LIN {X 0,Y 446.008,Z 588.455,A -85,B 0,C 180,E1 -8609.719,E2 -8609.719} C_VEL
LIN {X 0,Y 445.733,Z 595.064,A -85,B 0,C 180,E1 -8611.255,E2 -8611.255} C_VEL
LIN {X 0,Y 445.505,Z 599.999,A -85,B 0,C 180,E1 -8612.775,E2 -8612.775} C_VEL
LIN {X 0,Y 445.401,Z 603.162,A -85,B 0,C 180,E1 -8614.076,E2 -8614.076} C_VEL
LIN {X 0,Y 445.268,Z 605.906,A -85,B 0,C 180,E1 -8615.771,E2 -8615.771} C_VEL
LIN {X 0,Y 445.212,Z 606.838,A -85,B 0,C 180,E1 -8616.756,E2 -8616.756} C_VEL
LIN {X 0,Y 445.201,Z 607.248,A -85,B 0,C 180,E1 -8617.736,E2 -8617.736} C_VEL
LIN {X 0,Y 445.232,Z 607.217,A -85,B 0,C 180,E1 -8618.712,E2 -8618.712} C_VEL
LIN {X 0,Y 445.257,Z 606.684,A -85,B 0,C 180,E1 -8619.681,E2 -8619.681} C_VEL
LIN {X 0,Y 445.34,Z 604.85,A -85,B 0,C 180,E1 -8621.235,E2 -8621.235} C_VEL
LIN {X 0,Y 445.513,Z 601.175,A -85,B 0,C 180,E1 -8623.032,E2 -8623.032} C_VEL
LIN {X 0,Y 445.658,Z 596.958,A -85,B 0,C 180,E1 -8624.449,E2 -8624.449} C_VEL
LIN {X 0,Y 446.021,Z 590.447,A -85,B 0,C 180,E1 -8626.096,E2 -8626.096} C_VEL
LIN {X 0,Y 446.349,Z 583.463,A -85,B 0,C 180,E1 -8627.473,E2 -8627.473} C_VEL
LIN {X 0,Y 446.867,Z 574.417,A -85,B 0,C 180,E1 -8628.892,E2 -8628.892} C_VEL
LIN {X 0,Y 447.409,Z 565.251,A -85,B 0,C 180,E1 -8630.05,E2 -8630.05} C_VEL
LIN {X 0,Y 447.929,Z 555.119,A -85,B 0,C 180,E1 -8631.085,E2 -8631.085} C_VEL
LIN {X 0,Y 448.557,Z 543.89,A -85,B 0,C 180,E1 -8632.007,E2 -8632.007} C_VEL
LIN {X 0,Y 449.082,Z 532.298,A -85,B 0,C 180,E1 -8632.751,E2 -8632.751} C_VEL
LIN {X 0,Y 449.505,Z 519.239,A -85,B 0,C 180,E1 -8633.379,E2 -8633.379} C_VEL
LIN {X 0,Y 449.836,Z 507.364,A -85,B 0,C 180,E1 -8633.778,E2 -8633.778} C_VEL
LIN {X 0,Y 450.082,Z 490.19,A -85,B 0,C 180,E1 -8634.118,E2 -8634.118} C_VEL
LIN {X 0,Y 451.047,Z 413.44,A -85,B 0,C 180,E1 -8635.49,E2 -8635.49} C_VEL
LIN {X 0,Y 447.717,Z 396.497,A -85,B 0,C 180,E1 -8635.977,E2 -8635.977} C_VEL
LIN {X 0,Y 447.957,Z 383.895,A -85,B 0,C 180,E1 -8638.427,E2 -8638.427} C_VEL
LIN {X 0,Y 446.776,Z 375.836,A -85,B 0,C 180,E1 -8640.056,E2 -8640.056} C_VEL
LIN {X 0,Y 446.7,Z 375.846,A -85,B 0,C 180,E1 -8642.705,E2 -8642.705} C_VEL
LIN {X 0,Y 446.636,Z 375.853,A -85,B 0,C 180,E1 -8646.324,E2 -8646.324} C_VEL
LIN {X 0,Y 446.529,Z 375.863,A -85,B 0,C 180,E1 -8649.056,E2 -8649.056} C_VEL
LIN {X 0,Y 446.523,Z 375.865,A -85,B 0,C 180,E1 -8652.73,E2 -8652.73} C_VEL
LIN {X 0,Y 446.485,Z 375.87,A -85,B 0,C 180,E1 -8656.459,E2 -8656.459} C_VEL
LIN {X 0,Y 446.46,Z 375.871,A -85,B 0,C 180,E1 -8659.304,E2 -8659.304} C_VEL
LIN {X 0,Y 446.434,Z 375.876,A -85,B 0,C 180,E1 -8662.199,E2 -8662.199} C_VEL
LIN {X 0,Y 446.465,Z 375.869,A -85,B 0,C 180,E1 -8665.152,E2 -8665.152} C_VEL
LIN {X 0,Y 446.474,Z 375.87,A -85,B 0,C 180,E1 -8668.179,E2 -8668.179} C_VEL
LIN {X 0,Y 446.422,Z 375.878,A -85,B 0,C 180,E1 -8671.3,E2 -8671.3} C_VEL
LIN {X 0,Y 446.421,Z 375.874,A -85,B 0,C 180,E1 -8674.524,E2 -8674.524} C_VEL
LIN {X 0,Y 446.422,Z 375.875,A -85,B 0,C 180,E1 -8678.083,E2 -8678.083} C_VEL
LIN {X 0,Y 446.42,Z 375.877,A -85,B 0,C 180,E1 -8680.919,E2 -8680.919} C_VEL
LIN {X 0,Y 446.416,Z 375.875,A -85,B 0,C 180,E1 -8683.844,E2 -8683.844} C_VEL
LIN {X 0,Y 446.415,Z 375.874,A -85,B 0,C 180,E1 -8686.401,E2 -8686.401} C_VEL
LIN {X 0,Y 446.442,Z 375.872,A -85,B 0,C 180,E1 -8689.804,E2 -8689.804} C_VEL
LIN {X 0,Y 446.423,Z 375.874,A -85,B 0,C 180,E1 -8692.124,E2 -8692.124} C_VEL
LIN {X 0,Y 446.426,Z 375.876,A -85,B 0,C 180,E1 -8695.478,E2 -8695.478} C_VEL
LIN {X 0,Y 446.431,Z 375.879,A -85,B 0,C 180,E1 -8698.702,E2 -8698.702} C_VEL
LIN {X 0,Y 446.481,Z 375.868,A -85,B 0,C 180,E1 -8701.823,E2 -8701.823} C_VEL
LIN {X 0,Y 446.539,Z 376.057,A -85,B 0,C 180,E1 -8703.628,E2 -8703.628} C_VEL
LIN {X 0,Y 448.92,Z 388.648,A -85,B 0,C 180,E1 -8706.228,E2 -8706.228} C_VEL
LIN {X 0,Y 448.749,Z 396.065,A -85,B 0,C 180,E1 -8707.649,E2 -8707.649} C_VEL
LIN {X 0,Y 447.734,Z 415.115,A -85,B 0,C 180,E1 -8711.231,E2 -8711.231} C_VEL
LIN {X 0,Y 447.463,Z 420.329,A -85,B 0,C 180,E1 -8712.202,E2 -8712.202} C_VEL
LIN {X 0,Y 450.765,Z 442.467,A -85,B 0,C 180,E1 -8712.709,E2 -8712.709} C_VEL
LIN {X 0,Y 449.916,Z 528.45,A -85,B 0,C 180,E1 -8714.137,E2 -8714.137} C_VEL
LIN {X 0,Y 449.477,Z 541.635,A -85,B 0,C 180,E1 -8714.528,E2 -8714.528} C_VEL
LIN {X 0,Y 448.986,Z 554.347,A -85,B 0,C 180,E1 -8715.092,E2 -8715.092} C_VEL
LIN {X 0,Y 448.39,Z 566.46,A -85,B 0,C 180,E1 -8715.825,E2 -8715.825} C_VEL
LIN {X 0,Y 447.868,Z 576.888,A -85,B 0,C 180,E1 -8716.634,E2 -8716.634} C_VEL
LIN {X 0,Y 447.312,Z 587.338,A -85,B 0,C 180,E1 -8717.64,E2 -8717.64} C_VEL
LIN {X 0,Y 446.84,Z 596.026,A -85,B 0,C 180,E1 -8718.663,E2 -8718.663} C_VEL
LIN {X 0,Y 446.348,Z 604.028,A -85,B 0,C 180,E1 -8719.798,E2 -8719.798} C_VEL
LIN {X 0,Y 445.967,Z 611.859,A -85,B 0,C 180,E1 -8721.163,E2 -8721.163} C_VEL
LIN {X 0,Y 445.634,Z 619.035,A -85,B 0,C 180,E1 -8722.753,E2 -8722.753} C_VEL
LIN {X 0,Y 445.485,Z 623.252,A -85,B 0,C 180,E1 -8723.937,E2 -8723.937} C_VEL
LIN {X 0,Y 445.412,Z 627.473,A -85,B 0,C 180,E1 -8725.476,E2 -8725.476} C_VEL
LIN {X 0,Y 445.378,Z 629.359,A -85,B 0,C 180,E1 -8726.382,E2 -8726.382} C_VEL
LIN {X 0,Y 445.432,Z 630.779,A -85,B 0,C 180,E1 -8727.288,E2 -8727.288} C_VEL
LIN {X 0,Y 445.338,Z 632.395,A -85,B 0,C 180,E1 -8729.097,E2 -8729.097} C_VEL
LIN {X 0,Y 445.342,Z 632.616,A -85,B 0,C 180,E1 -8730.001,E2 -8730.001} C_VEL
LIN {X 0,Y 445.338,Z 632.4,A -85,B 0,C 180,E1 -8730.905,E2 -8730.905} C_VEL
LIN {X 0,Y 445.433,Z 630.78,A -85,B 0,C 180,E1 -8732.714,E2 -8732.714} C_VEL
LIN {X 0,Y 445.379,Z 629.368,A -85,B 0,C 180,E1 -8733.62,E2 -8733.62} C_VEL
LIN {X 0,Y 445.476,Z 626.406,A -85,B 0,C 180,E1 -8734.979,E2 -8734.979} C_VEL
LIN {X 0,Y 445.575,Z 620.951,A -85,B 0,C 180,E1 -8736.749,E2 -8736.749} C_VEL
LIN {X 0,Y 445.792,Z 615.209,A -85,B 0,C 180,E1 -8738.158,E2 -8738.158} C_VEL
LIN {X 0,Y 446.137,Z 608.248,A -85,B 0,C 180,E1 -8739.522,E2 -8739.522} C_VEL
LIN {X 0,Y 446.576,Z 599.533,A -85,B 0,C 180,E1 -8740.887,E2 -8740.887} C_VEL
LIN {X 0,Y 447.171,Z 590.606,A -85,B 0,C 180,E1 -8742.021,E2 -8742.021} C_VEL
LIN {X 0,Y 447.705,Z 580.034,A -85,B 0,C 180,E1 -8743.118,E2 -8743.118} C_VEL
LIN {X 0,Y 448.321,Z 568.493,A -85,B 0,C 180,E1 -8744.064,E2 -8744.064} C_VEL
LIN {X 0,Y 448.966,Z 556.065,A -85,B 0,C 180,E1 -8744.853,E2 -8744.853} C_VEL
LIN {X 0,Y 449.473,Z 544.263,A -85,B 0,C 180,E1 -8745.416,E2 -8745.416} C_VEL
LIN {X 0,Y 449.902,Z 531.477,A -85,B 0,C 180,E1 -8745.837,E2 -8745.837} C_VEL
LIN {X 0,Y 450.252,Z 513.687,A -85,B 0,C 180,E1 -8746.173,E2 -8746.173} C_VEL
LIN {X 0,Y 450.851,Z 440.892,A -85,B 0,C 180,E1 -8747.381,E2 -8747.381} C_VEL
LIN {X 0,Y 447.474,Z 419.812,A -85,B 0,C 180,E1 -8747.898,E2 -8747.898} C_VEL
LIN {X 0,Y 448.378,Z 402.59,A -85,B 0,C 180,E1 -8751.132,E2 -8751.132} C_VEL
LIN {X 0,Y 449.121,Z 390.1,A -85,B 0,C 180,E1 -8753.519,E2 -8753.519} C_VEL
LIN {X 0,Y 447.614,Z 381.351,A -85,B 0,C 180,E1 -8755.332,E2 -8755.332} C_VEL
LIN {X 0,Y 446.492,Z 375.869,A -85,B 0,C 180,E1 -8756.516,E2 -8756.516} C_VEL
LIN {X 0,Y 446.455,Z 375.878,A -85,B 0,C 180,E1 -8759.21,E2 -8759.21} C_VEL
LIN {X 0,Y 446.428,Z 375.876,A -85,B 0,C 180,E1 -8762.362,E2 -8762.362} C_VEL
LIN {X 0,Y 446.425,Z 375.878,A -85,B 0,C 180,E1 -8765.627,E2 -8765.627} C_VEL
LIN {X 0,Y 446.461,Z 375.876,A -85,B 0,C 180,E1 -8769.026,E2 -8769.026} C_VEL
LIN {X 0,Y 446.44,Z 375.874,A -85,B 0,C 180,E1 -8772.278,E2 -8772.278} C_VEL
LIN {X 0,Y 446.459,Z 375.875,A -85,B 0,C 180,E1 -8775.104,E2 -8775.104} C_VEL
LIN {X 0,Y 446.433,Z 375.876,A -85,B 0,C 180,E1 -8778.609,E2 -8778.609} C_VEL
LIN {X 0,Y 446.447,Z 375.877,A -85,B 0,C 180,E1 -8780.973,E2 -8780.973} C_VEL
LIN {X 0,Y 446.424,Z 375.875,A -85,B 0,C 180,E1 -8784.374,E2 -8784.374} C_VEL
LIN {X 0,Y 446.428,Z 375.873,A -85,B 0,C 180,E1 -8787.639,E2 -8787.639} C_VEL
LIN {X 0,Y 446.454,Z 375.875,A -85,B 0,C 180,E1 -8790.791,E2 -8790.791} C_VEL
LIN {X 0,Y 446.484,Z 375.862,A -85,B 0,C 180,E1 -8793.849,E2 -8793.849} C_VEL
LIN {X 0,Y 446.432,Z 375.871,A -85,B 0,C 180,E1 -8796.823,E2 -8796.823} C_VEL
LIN {X 0,Y 446.45,Z 375.871,A -85,B 0,C 180,E1 -8799.737,E2 -8799.737} C_VEL
LIN {X 0,Y 446.468,Z 375.873,A -85,B 0,C 180,E1 -8802.597,E2 -8802.597} C_VEL
LIN {X 0,Y 446.475,Z 375.861,A -85,B 0,C 180,E1 -8805.413,E2 -8805.413} C_VEL
LIN {X 0,Y 446.523,Z 375.866,A -85,B 0,C 180,E1 -8808.193,E2 -8808.193} C_VEL
LIN {X 0,Y 446.606,Z 375.854,A -85,B 0,C 180,E1 -8811.858,E2 -8811.858} C_VEL
LIN {X 0,Y 446.651,Z 375.848,A -85,B 0,C 180,E1 -8814.583,E2 -8814.583} C_VEL
LIN {X 0,Y 446.67,Z 375.848,A -85,B 0,C 180,E1 -8818.197,E2 -8818.197} C_VEL
LIN {X 0,Y 446.798,Z 375.83,A -85,B 0,C 180,E1 -8820,E2 -8820} C_VEL
LIN {X 0,Y 446.697,Z 375.84,A -85,B 0,C 180,E1 -8822.705,E2 -8822.705} C_VEL
LIN {X 0,Y 446.653,Z 375.846,A -85,B 0,C 180,E1 -8826.324,E2 -8826.324} C_VEL
LIN {X 0,Y 446.544,Z 375.859,A -85,B 0,C 180,E1 -8829.055,E2 -8829.055} C_VEL
LIN {X 0,Y 446.528,Z 375.861,A -85,B 0,C 180,E1 -8832.73,E2 -8832.73} C_VEL
LIN {X 0,Y 446.502,Z 375.867,A -85,B 0,C 180,E1 -8836.228,E2 -8836.228} C_VEL
LIN {X 0,Y 446.476,Z 375.872,A -85,B 0,C 180,E1 -8839.303,E2 -8839.303} C_VEL
LIN {X 0,Y 446.424,Z 375.877,A -85,B 0,C 180,E1 -8842.199,E2 -8842.199} C_VEL
LIN {X 0,Y 446.45,Z 375.876,A -85,B 0,C 180,E1 -8845.153,E2 -8845.153} C_VEL
LIN {X 0,Y 446.491,Z 375.868,A -85,B 0,C 180,E1 -8848.178,E2 -8848.178} C_VEL
LIN {X 0,Y 446.515,Z 375.874,A -85,B 0,C 180,E1 -8849.205,E2 -8849.205} C_VEL
LIN {X 0,Y 448.283,Z 385.967,A -85,B 0,C 180,E1 -8851.643,E2 -8851.643} C_VEL
LIN {X 0,Y 447.748,Z 397.339,A -85,B 0,C 180,E1 -8854.191,E2 -8854.191} C_VEL
LIN {X 0,Y 451.088,Z 414.15,A -85,B 0,C 180,E1 -8854.624,E2 -8854.624} C_VEL
LIN {X 0,Y 450.084,Z 504.878,A -85,B 0,C 180,E1 -8856.15,E2 -8856.15} C_VEL
LIN {X 0,Y 449.747,Z 517.792,A -85,B 0,C 180,E1 -8856.548,E2 -8856.548} C_VEL
LIN {X 0,Y 449.312,Z 530.874,A -85,B 0,C 180,E1 -8857.147,E2 -8857.147} C_VEL
LIN {X 0,Y 448.825,Z 541.762,A -85,B 0,C 180,E1 -8857.819,E2 -8857.819} C_VEL
LIN {X 0,Y 448.191,Z 553.201,A -85,B 0,C 180,E1 -8858.72,E2 -8858.72} C_VEL
LIN {X 0,Y 447.644,Z 563.236,A -85,B 0,C 180,E1 -8859.708,E2 -8859.708} C_VEL
LIN {X 0,Y 447.011,Z 573.19,A -85,B 0,C 180,E1 -8860.921,E2 -8860.921} C_VEL
LIN {X 0,Y 446.543,Z 582.158,A -85,B 0,C 180,E1 -8862.291,E2 -8862.291} C_VEL
LIN {X 0,Y 446.1,Z 588.864,A -85,B 0,C 180,E1 -8863.555,E2 -8863.555} C_VEL
LIN {X 0,Y 445.831,Z 594.286,A -85,B 0,C 180,E1 -8864.815,E2 -8864.815} C_VEL
LIN {X 0,Y 445.618,Z 598.585,A -85,B 0,C 180,E1 -8866.056,E2 -8866.056} C_VEL
LIN {X 0,Y 445.436,Z 603.236,A -85,B 0,C 180,E1 -8867.865,E2 -8867.865} C_VEL
LIN {X 0,Y 445.306,Z 605.604,A -85,B 0,C 180,E1 -8869.25,E2 -8869.25} C_VEL
LIN {X 0,Y 445.243,Z 607.118,A -85,B 0,C 180,E1 -8870.846,E2 -8870.846} C_VEL
LIN {X 0,Y 445.219,Z 607.459,A -85,B 0,C 180,E1 -8872.118,E2 -8872.118} C_VEL
LIN {X 0,Y 445.235,Z 606.828,A -85,B 0,C 180,E1 -8873.614,E2 -8873.614} C_VEL
LIN {X 0,Y 445.366,Z 604.658,A -85,B 0,C 180,E1 -8875.382,E2 -8875.382} C_VEL
LIN {X 0,Y 445.543,Z 600.895,A -85,B 0,C 180,E1 -8877.152,E2 -8877.152} C_VEL
LIN {X 0,Y 445.743,Z 596.32,A -85,B 0,C 180,E1 -8878.646,E2 -8878.646} C_VEL
LIN {X 0,Y 445.996,Z 590.621,A -85,B 0,C 180,E1 -8880.077,E2 -8880.077} C_VEL
LIN {X 0,Y 446.391,Z 583.146,A -85,B 0,C 180,E1 -8881.558,E2 -8881.558} C_VEL
LIN {X 0,Y 446.859,Z 574.839,A -85,B 0,C 180,E1 -8882.863,E2 -8882.863} C_VEL
LIN {X 0,Y 447.419,Z 565.688,A -85,B 0,C 180,E1 -8884.032,E2 -8884.032} C_VEL
LIN {X 0,Y 447.923,Z 557.075,A -85,B 0,C 180,E1 -8884.938,E2 -8884.938} C_VEL
